(* Vertikale Linie zeichnen *)
IF Iin_X1 = Iin_X2 THEN
	in_Offset_1 := (Iin_Y1 * 80) + Iin_X1;
	FOR in_ROW_Index := Iin_Y1 TO Iin_Y2 DO
		by_old_Char := Xus_TN_SCREEN.bya_CHAR[in_Offset_1]; (* bestehendes Zeichen auslesen *)
		by_Char := by_Vertikal_Line_Char; (* Standardzeichen vorbelegen *)
		IF by_old_Char = by_Horzontal_Line_Char THEN (* Schnittpunkt erkannt *)
			IF in_ROW_Index = Iin_Y1 THEN (* Anfang der Linie behandeln *)
				by_Char := by_Connect_Top_Char;
			ELSIF in_ROW_Index = Iin_Y2 THEN (* Ende der Linie behandeln *)
				by_Char := by_Connect_Bottom_Char;
			ELSE (* Kreuzungspunkt behandeln *)
				by_Char := by_Connect_Cruz_Char;
			END_IF;
		END_IF;
		Xus_TN_SCREEN.bya_Line_Update[in_ROW_Index] := TRUE; (* Zeile zum Updaten freigeben *)
		Xus_TN_SCREEN.bya_CHAR[in_Offset_1] := by_Char;
		Xus_TN_SCREEN.bya_COLOR[in_Offset_1] := Iby_Attr;
		in_Offset_1 := in_Offset_1 + 80;
	END_FOR;

ELSIF Iin_Y1 = Iin_Y2 THEN (* Horzontale Linie zeichnen *)
	Xus_TN_SCREEN.bya_Line_Update[Iin_Y1] := TRUE; (* Zeile zum Updaten freigeben *)
	in_Offset_1 := (Iin_Y1 * 80) + Iin_X1;
	FOR in_COL_Index := Iin_X1 TO Iin_X2 DO
		by_old_Char := Xus_TN_SCREEN.bya_CHAR[in_Offset_1]; (* bestehendes Zeichen auslesen *)
		by_Char := by_Horzontal_Line_Char; (* Standardzeichen vorbelegen *)
		IF by_old_Char = by_Vertikal_Line_Char THEN (* Schnittpunkt erkannt *)
			IF in_COL_Index = Iin_X1 THEN (* Anfang der Linie behandeln *)
				by_Char := by_Connect_Left_Char;
			ELSIF in_COL_Index = Iin_X2 THEN (* Ende der Linie behandeln *)
				by_Char := by_Connect_Right_Char;
			ELSE (* Kreuzungspunkt behandeln *)
				by_Char := by_Connect_Cruz_Char;
			END_IF;
		END_IF;
		Xus_TN_SCREEN.bya_CHAR[in_Offset_1] := by_Char;
		Xus_TN_SCREEN.bya_COLOR[in_Offset_1] := Iby_Attr;
		in_Offset_1 := in_Offset_1 + 1;
	END_FOR;
END_IF;

(* revision history
ks	10. mai. 2010	rev 1.0
	original version
*)
END_FUNCTION_BLOCK

(* POU TN_SC_ADD_SHADOW, ST *)
FUNCTION_BLOCK TN_SC_ADD_SHADOW
VAR
	in_Offset : INT;
	in_X : INT;
	in_Y : INT;
END_VAR
VAR_INPUT
	Iin_Y1 : INT;
	Iin_X1 : INT;
	Iin_Y2 : INT;
	Iin_X2 : INT;
	Iin_OPTION : INT;
END_VAR
VAR_IN_OUT
	Xus_TN_SCREEN : us_TN_SCREEN;
END_VAR

(*
version 1.0		10. mai 2010
programmer		ks
tested by		ks

TN_SC_ADD_SHADOW zeichnet auf der linken und unteren Seite eines rechteckigen Bereiches einen Schatten
*)
IF TN_SC_XY2_ERROR(Iin_X1,Iin_Y1,Iin_X2,Iin_Y2) THEN RETURN; END_IF;

IF Iin_Y1 < 0 OR Iin_X1 < 0 OR Iin_Y2 < 0 OR Iin_X2 < 0 THEN RETURN; END_IF; (* min werte prüfen *)
IF Iin_Y1 > 23 OR Iin_X1 > 79 OR Iin_Y2 > 23 OR Iin_X2 > 79 THEN RETURN; END_IF; (* max werte prüfen *)

in_Offset := (Iin_Y1 * 80) + Iin_X2;

IF Iin_OPTION = INT#00 THEN
	(* Schatten durch Farbanpassung erzeugen *)
	FOR in_Y := Iin_Y1 TO Iin_Y2 DO
		Xus_TN_SCREEN.bya_COLOR[in_Offset] := TN_SC_SHADOW_ATTR(Xus_TN_SCREEN.bya_COLOR[in_Offset]);
		in_Offset := in_Offset + 80;
		Xus_TN_SCREEN.bya_Line_Update[in_Y] := TRUE; (* Zeile für Update eintragen *)
	END_FOR;
ELSE
	(* Schatten durch Farbe Schwarz und Leerzeichen erzeugen *)
	FOR in_Y := Iin_Y1 TO Iin_Y2 DO
		Xus_TN_SCREEN.bya_COLOR[in_Offset] := BYTE#00;
		Xus_TN_SCREEN.bya_CHAR[in_Offset] := BYTE#32;
		in_Offset := in_Offset + 80;
		Xus_TN_SCREEN.bya_Line_Update[in_Y] := TRUE; (* Zeile für Update eintragen *)
	END_FOR;
END_IF;

in_Offset := (Iin_Y2 * 80) + Iin_X1;

IF Iin_OPTION = INT#00 THEN
	(* Schatten durch Farbanpassung erzeugen *)
	FOR in_X  := Iin_X1 TO Iin_X2 DO
		Xus_TN_SCREEN.bya_COLOR[in_Offset] := TN_SC_SHADOW_ATTR(Xus_TN_SCREEN.bya_COLOR[in_Offset]);
		in_Offset := in_Offset + 1;
	END_FOR;
ELSE
	(* Schatten durch Farbe Schwarz und Leerzeichen erzeugen *)
	FOR in_X  := Iin_X1 TO Iin_X2 DO
		Xus_TN_SCREEN.bya_COLOR[in_Offset] := BYTE#00;
		Xus_TN_SCREEN.bya_CHAR[in_Offset] := BYTE#32;
		in_Offset := in_Offset + 1;
	END_FOR;
END_IF;

(* revision history
ks	10. mai. 2010	rev 1.0
	original version
*)
END_FUNCTION_BLOCK

(* POU TN_SC_SHADOW_ATTR, ST *)
FUNCTION TN_SC_SHADOW_ATTR : BYTE
VAR_INPUT
	Iby_ATTR : BYTE;
END_VAR

(*
version 1.0		10. mai 2010
programmer		ks
tested by		ks

TN_SC_SHADOW_ATTR berechnet aus einem normalen einem abgedunkelten Farbcode
*)
(* Background Farbe auf Schwarz ändern      *)
(* und dunkle Fordergrundfarben einschalten *)  
TN_SC_SHADOW_ATTR := ((Iby_ATTR AND BYTE#2#11110000) OR BYTE#2#00001000);

(* revision history
ks	10. mai. 2010	rev 1.0
	original version
*)
END_FUNCTION

(* POU TN_SC_BOX, ST *)
FUNCTION_BLOCK TN_SC_BOX
VAR
	FB_TN_SC_FILL : TN_SC_FILL;
	by_BorderChar_L_T : BYTE;
	by_BorderChar_T : BYTE;
	by_BorderChar_B : BYTE;
	by_BorderChar_R_T : BYTE;
	by_BorderChar_L : BYTE;
	by_BorderChar_R : BYTE;
	by_BorderChar_L_B : BYTE;
	by_BorderChar_R_B : BYTE;
	in_Y : INT;
	in_X : INT;
	in_Border_Offset : INT;
	in_Offset_1 : INT;
	in_Offset_2 : INT;
END_VAR
VAR_INPUT
	Iin_Y1 : INT;
	Iin_X1 : INT;
	Iin_Y2 : INT;
	Iin_X2 : INT;
	Iby_FILL : BYTE;
	Iby_ATTR : BYTE;
	Iin_BORDER : INT;
END_VAR
VAR_IN_OUT
	Xus_TN_SCREEN : us_TN_SCREEN;
END_VAR

(*
version 1.0		10. mai 2010
programmer		ks
tested by		ks

TN_SC_BOX füllt einen rechteckigen Bereich mit einem Zeichen und zeichnet eine Umrandung
*)
IF TN_SC_XY2_ERROR(Iin_X1,Iin_Y1,Iin_X2,Iin_Y2) THEN RETURN; END_IF;

(* Bordertype bestimmen *)
CASE Iin_Border OF
0:
	in_Border_Offset := 0;
1:
	by_BorderChar_L_T := BYTE#218; (* links oben *)
	by_BorderChar_T := BYTE#196; (* oben *)
	by_BorderChar_R_T := BYTE#191; (* rechts oben *)
	by_BorderChar_L := BYTE#179; (* links *)
	by_BorderChar_R := BYTE#179; (* rechts *)
	by_BorderChar_B := BYTE#196; (* unten *)
	by_BorderChar_L_B := BYTE#217; (* links unten *)
	by_BorderChar_R_B := BYTE#192; (* rechts unten *)
	in_Border_Offset := 1;
 2:
	by_BorderChar_L_T := BYTE#201;
	by_BorderChar_T := BYTE#205;
	by_BorderChar_R_T := BYTE#187;
	by_BorderChar_L := BYTE#186;
	by_BorderChar_R := BYTE#186;
	by_BorderChar_B := BYTE#205;
	by_BorderChar_L_B := BYTE#188;
	by_BorderChar_R_B := BYTE#200;
	in_Border_Offset := 1;
ELSE
	by_BorderChar_L_T := BYTE#32;
	by_BorderChar_T := BYTE#32;
	by_BorderChar_R_T := BYTE#32;
	by_BorderChar_L := BYTE#32;
	by_BorderChar_R := BYTE#32;
	by_BorderChar_B := BYTE#32;
	by_BorderChar_L_B := BYTE#32;
	by_BorderChar_R_B := BYTE#32;
	in_Border_Offset := 1;

END_CASE;

IF Iby_FILL > BYTE#0 THEN (* FILL Zeichen vorhanden ? -> Box zeichnen *)

	(* Fill-Function um eine Zeichenreihe kleiner zeichnen *)
	FB_TN_SC_FILL(	Iin_Y1 := Iin_Y1 + in_Border_Offset,
					Iin_X1 := Iin_X1 + in_Border_Offset,
					Iin_Y2 := Iin_Y2 - in_Border_Offset,
					Iin_X2 := Iin_X2 - in_Border_Offset,
					Iby_CHAR := Iby_FILL,
					Iby_Attr := Iby_ATTR,
					Xus_TN_SCREEN := Xus_TN_SCREEN);
END_IF;

IF Iin_BORDER = 0 THEN RETURN; END_IF;

(* linken und rechten Rand ausgeben *)

in_Offset_1 := (Iin_Y1 * 80) + Iin_X1;
in_Offset_2 := (Iin_Y1 * 80) + Iin_X2;

FOR in_Y := Iin_Y1 TO Iin_Y2 DO

	(* Zeile zum Updaten freigeben *)
	Xus_TN_SCREEN.bya_Line_Update[in_Y] := TRUE;

	Xus_TN_SCREEN.bya_CHAR[in_Offset_1] := by_BorderChar_L;
	Xus_TN_SCREEN.bya_COLOR[in_Offset_1] := Iby_Attr;

	Xus_TN_SCREEN.bya_CHAR[in_Offset_2] := by_BorderChar_R;
	Xus_TN_SCREEN.bya_COLOR[in_Offset_2] := Iby_Attr;

	in_Offset_1 := in_Offset_1 + 80;
	in_Offset_2 := in_Offset_2 + 80;

END_FOR;

(* unteren und oberen Rand ausgeben *)
in_Offset_1 := (Iin_Y1 * 80) + Iin_X1;
in_Offset_2 := (Iin_Y2 * 80) + Iin_X1;

FOR in_X := Iin_X1 TO Iin_X2 DO

	Xus_TN_SCREEN.bya_CHAR[in_Offset_1] := by_BorderChar_T;
	Xus_TN_SCREEN.bya_COLOR[in_Offset_1] := Iby_Attr;

	Xus_TN_SCREEN.bya_CHAR[in_Offset_2] := by_BorderChar_B;
	Xus_TN_SCREEN.bya_COLOR[in_Offset_2] := Iby_Attr;

	in_Offset_1 := in_Offset_1 + INT#1;
	in_Offset_2 := in_Offset_2 + INT#1;

END_FOR;

(* linke obere Ecke ausgeben *)
in_Offset_1 := (Iin_Y1 * 80) + Iin_X1;
Xus_TN_SCREEN.bya_CHAR[in_Offset_1] := by_BorderChar_L_T;
Xus_TN_SCREEN.bya_COLOR[in_Offset_1] := Iby_Attr;

(* rechte obere Ecke ausgeben *)
in_Offset_1 := (Iin_Y1 * 80) + Iin_X2;
Xus_TN_SCREEN.bya_CHAR[in_Offset_1] := by_BorderChar_R_T;
Xus_TN_SCREEN.bya_COLOR[in_Offset_1] := Iby_Attr;

(* linke untere Ecke ausgeben *)
in_Offset_1 := (Iin_Y2 * 80) + Iin_X1;
Xus_TN_SCREEN.bya_CHAR[in_Offset_1] := by_BorderChar_R_B;
Xus_TN_SCREEN.bya_COLOR[in_Offset_1] := Iby_Attr;

(* rechte untere Ecke ausgeben *)
in_Offset_1 := (Iin_Y2 * 80) + Iin_X2;
Xus_TN_SCREEN.bya_CHAR[in_Offset_1] := by_BorderChar_L_B;
Xus_TN_SCREEN.bya_COLOR[in_Offset_1] := Iby_Attr;

(* revision history
ks	10. mai. 2010	rev 1.0
	original version
*)
END_FUNCTION_BLOCK

(* POU TN_SC_FILL, ST *)
FUNCTION_BLOCK TN_SC_FILL
VAR
	in_X : INT;
	in_Y : INT;
	in_Offset : INT;
END_VAR
VAR_INPUT
	Iin_Y1 : INT;
	Iin_X1 : INT;
	Iin_Y2 : INT;
	Iin_X2 : INT;
	Iby_CHAR : BYTE;
	Iby_Attr : BYTE;
END_VAR
VAR_IN_OUT
	Xus_TN_SCREEN : us_TN_SCREEN;
END_VAR

(*
version 1.0		10. mai 2010
programmer		ks
tested by		ks

TN_SC_FILL füllt einen rechteckigen Bereich mit einem Zeichen
*)
IF TN_SC_XY2_ERROR(Iin_X1,Iin_Y1,Iin_X2,Iin_Y2) THEN RETURN; END_IF;

FOR in_Y := Iin_Y1 TO Iin_Y2 DO
	Xus_TN_SCREEN.bya_Line_Update[in_Y] := TRUE; (* Zeile zum Updaten freigeben *)
	in_Offset := (in_Y * 80) + Iin_X1;
	FOR in_X := Iin_X1 TO Iin_X2 DO
		Xus_TN_SCREEN.bya_CHAR[in_Offset]  := Iby_CHAR; (* Zeichen eintragen *)
		Xus_TN_SCREEN.bya_COLOR[in_Offset] := Iby_Attr; (* Farbe eintragen *)
		in_Offset := in_Offset + 1;
	END_FOR;
END_FOR;

(* revision history
ks	10. mai. 2010	rev 1.0
	original version
*)
END_FUNCTION_BLOCK

(* POU TN_SC_WRITE_C, ST *)
FUNCTION_BLOCK TN_SC_WRITE_C
VAR
	FB_TN_SC_WRITE : TN_SC_WRITE;
END_VAR
VAR_INPUT
	Iin_Y : INT;
	Iin_X : INT;
	Iby_ATTR : BYTE;
	Ist_STRING : STRING;
	Iin_LENGTH : INT;
	Iin_OPTION : INT;
END_VAR
VAR_IN_OUT
	Xus_TN_SCREEN : us_TN_SCREEN;
END_VAR

(*
version 1.0		10. mai 2010
programmer		ks
tested by		ks

TN_SC_WRITE_C korrigiert die Textlänge und schreibt den Text an die angegebenen Koordinate
*)
(* Text ausgeben *)
FB_TN_SC_WRITE( Iin_Y := Iin_Y,
				Iin_X := Iin_X,
				Iby_ATTR := Iby_ATTR,
				Ist_STRING := FIX(str:=Ist_STRING,L:=Iin_LENGTH,C:=BYTE#32,M:=Iin_OPTION),
				Xus_TN_SCREEN := Xus_TN_SCREEN);

(* revision history
ks	10. mai. 2010	rev 1.0
	original version
*)
END_FUNCTION_BLOCK

(* POU TN_SC_WRITE, ST *)
FUNCTION_BLOCK TN_SC_WRITE
VAR
	bo_Color : BOOL;
	in_Offset : INT;
	in_Char_Index : INT;
	in_String_Length : INT;
END_VAR
VAR_INPUT
	Iin_Y : INT;
	Iin_X : INT;
	Iby_ATTR : BYTE;
	Ist_STRING : STRING;
END_VAR
VAR_IN_OUT
	Xus_TN_SCREEN : us_TN_SCREEN;
END_VAR

(*
version 1.0		10. mai 2010
programmer		ks
tested by		ks

TN_SC_WRITE schreibt einem Text an die angegebene Koordinate
*)
in_String_Length := LEN(Ist_STRING);
IF TN_SC_XY_ERROR(Iin_X + in_String_Length - 1,Iin_Y) THEN RETURN; END_IF;
Xus_TN_SCREEN.bya_Line_Update[Iin_Y] := TRUE; (* Zeile zum Updaten freigeben *)
in_Offset := (Iin_Y * 80) + Iin_X; (* Offset des ersten Zeichen berechnen *)
bo_Color := Iby_ATTR <> BYTE#00;

(* Zeichen und Attribute des String kopieren *)
FOR in_Char_Index := 1 TO in_String_Length DO
	IF bo_Color THEN Xus_TN_SCREEN.bya_COLOR[in_Offset] := Iby_ATTR; END_IF;
	Xus_TN_SCREEN.bya_CHAR[in_Offset] := CODE(STR:=Ist_STRING,POS:=in_Char_Index);
	in_Offset := in_Offset + INT#1;
END_FOR;

Xus_TN_SCREEN.in_EOS_Offset := in_Offset; (* End of String Offset sichern *)

(* revision history
ks	10. mai. 2010	rev 1.0
	original version
*)
END_FUNCTION_BLOCK

(* POU TN_SC_XY_ERROR, ST *)
FUNCTION TN_SC_XY_ERROR : BOOL
VAR_INPUT
	X : INT;
	Y : INT;
END_VAR

(*
version 1.0		10. mai 2010
programmer		ks
tested by		ks

TN_SC_XY_ERROR prüft ob die angegenene Koordinaten gültig sind 
*)
(* min und max werte prüfen *)
TN_SC_XY_ERROR := Y < 0 OR X < 0 OR Y > 23 OR X > 79;

(* revision history
ks	10. mai. 2010	rev 1.0
	original version
*)
END_FUNCTION

(* POU TN_INPUT_SELECT_TEXT, ST *)
FUNCTION_BLOCK TN_INPUT_SELECT_TEXT
VAR
	in_count : INT;
	by_Attr : BYTE;
	st_String : STRING;
END_VAR
VAR
	FB_TN_SC_WRITE : TN_SC_WRITE;
END_VAR
VAR_IN_OUT
	Xus_TN_SCREEN : us_TN_SCREEN;
	Xus_TN_INPUT_CONTROL_DATA : us_TN_INPUT_CONTROL_DATA;
END_VAR

(*
version 1.1		06. apr 2011
programmer		ks
tested by			ks

TN_SELECT_TEXT dient zur verwaltung und darstellung einer Elementeauswahl
*)
(* Benutzereingabe auswerten -> Selektion Text n *)
IF Xus_TN_INPUT_CONTROL_DATA.bo_Focus = TRUE THEN

(* Leertaste-Taste auswerten *)
	IF Xus_TN_INPUT_CONTROL_DATA.by_Input_ASCII_Code = BYTE#32 THEN
		Xus_TN_INPUT_CONTROL_DATA.in_selected := Xus_TN_INPUT_CONTROL_DATA.in_selected + INT#01; 
		Xus_TN_INPUT_CONTROL_DATA.bo_Update_Input := TRUE;
	END_IF;
 
	(* Return-Taste auswerten *)
	IF Xus_TN_INPUT_CONTROL_DATA.by_Input_Exten_Code = BYTE#13 THEN
		Xus_TN_INPUT_CONTROL_DATA.bo_Input_Entered := TRUE;
	END_IF;

END_IF;

(* Aktualisierung der Anzeige *)
IF (Xus_TN_INPUT_CONTROL_DATA.bo_Update_Input = TRUE) OR (Xus_TN_INPUT_CONTROL_DATA.bo_Update_All = TRUE) THEN

	(* Title-Text ausgeben *)
	IF Xus_TN_INPUT_CONTROL_DATA.bo_Update_All = TRUE THEN

		IF (Xus_TN_INPUT_CONTROL_DATA.in_Title_X_Offset = INT#00) AND (Xus_TN_INPUT_CONTROL_DATA.in_Title_Y_Offset = INT#00) THEN
			(* wenn Offset X,Y =0 dann Titlestring links vom Element positionieren *)
			FB_TN_SC_WRITE.Iin_Y := Xus_TN_INPUT_CONTROL_DATA.in_Y;
			FB_TN_SC_WRITE.Iin_X := Xus_TN_INPUT_CONTROL_DATA.in_X - LEN(Xus_TN_INPUT_CONTROL_DATA.st_Title_String);

		ELSE
			(* Title-Text durch Row, Color-Offset ausgeben *)
			FB_TN_SC_WRITE.Iin_Y := Xus_TN_INPUT_CONTROL_DATA.in_Y + Xus_TN_INPUT_CONTROL_DATA.in_Title_Y_Offset;
			FB_TN_SC_WRITE.Iin_X := Xus_TN_INPUT_CONTROL_DATA.in_X + Xus_TN_INPUT_CONTROL_DATA.in_Title_X_Offset;
		END_IF;

		(* Title-Text durch Row, Color-Offset ausgeben *)
		FB_TN_SC_WRITE(	Iby_ATTR := Xus_TN_INPUT_CONTROL_DATA.by_Title_Attr,
						Ist_STRING := Xus_TN_INPUT_CONTROL_DATA.st_Title_String,
						Xus_TN_SCREEN := Xus_TN_SCREEN);

	END_IF;

	(* Eingabezeile verarbeiten *)

	(* Anzahl der Elemente bestimmen *)
	in_count := ELEMENT_COUNT(SEP:=BYTE#35,ELEMENT:=Xus_TN_INPUT_CONTROL_DATA.st_Input_Data);

	IF in_Count > INT#00 THEN

		IF Xus_TN_INPUT_CONTROL_DATA.in_selected < INT#1 THEN
			Xus_TN_INPUT_CONTROL_DATA.in_selected := INT#01;
		END_IF;

		IF Xus_TN_INPUT_CONTROL_DATA.in_selected > in_count THEN
			Xus_TN_INPUT_CONTROL_DATA.in_selected := INT#01;
		END_IF;

		st_String := ELEMENT_GET(SEP:=BYTE#35,POS:=Xus_TN_INPUT_CONTROL_DATA.in_selected - 1,ELEMENT:=Xus_TN_INPUT_CONTROL_DATA.st_Input_Data);

		st_String := FIX(	str:=st_String,
							L:=LEN(Xus_TN_INPUT_CONTROL_DATA.st_Input_Mask),
							C:=BYTE#32,
							M:=Xus_TN_INPUT_CONTROL_DATA.in_Input_Option);

		Xus_TN_INPUT_CONTROL_DATA.st_Input_String := st_String;

		IF Xus_TN_INPUT_CONTROL_DATA.bo_Focus = TRUE THEN
			by_Attr := Xus_TN_INPUT_CONTROL_DATA.by_Attr_mF;
		ELSE
			by_Attr := Xus_TN_INPUT_CONTROL_DATA.by_Attr_oF;
		END_IF;

		FB_TN_SC_WRITE(	Iin_Y := Xus_TN_INPUT_CONTROL_DATA.in_Y,
						Iin_X := Xus_TN_INPUT_CONTROL_DATA.in_X,
						Iby_ATTR := by_Attr,
						Ist_STRING := st_String,
						Xus_TN_SCREEN := Xus_TN_SCREEN);
	END_IF;

	(* Cursor auf aktuelle Position setzen *)
	Xus_TN_INPUT_CONTROL_DATA.in_Cursor_Y := Xus_TN_INPUT_CONTROL_DATA.in_Y;
	Xus_TN_INPUT_CONTROL_DATA.in_Cursor_X := Xus_TN_INPUT_CONTROL_DATA.in_X;

	(* Update-Flag's rücksetzen *)
	Xus_TN_INPUT_CONTROL_DATA.bo_Update_All := FALSE;
	Xus_TN_INPUT_CONTROL_DATA.bo_Update_Input := FALSE;

END_IF;

(* revision history

ks	06. apr. 2011	rev 1.1
	list_len und list_get durch element_count und element_get ersetzt

ks	10. mai. 2010	rev 1.0
	original version
*)
END_FUNCTION_BLOCK

(* POU TN_INPUT_EDIT_LINE, ST *)
FUNCTION_BLOCK TN_INPUT_EDIT_LINE
VAR
	in_count : INT;
	in_Count_End : INT;
	in_CursorOffset : INT;
	by_Attr : BYTE;
	st_String : STRING;
	bo_Pos_Found : BOOL;
	st_CHAR : STRING(1);
	in_old_charpos : INT;
END_VAR
VAR
	FB_TN_SC_WRITE : TN_SC_WRITE;
END_VAR
VAR_IN_OUT
	Xus_TN_SCREEN : us_TN_SCREEN;
	Xus_TN_INPUT_CONTROL_DATA : us_TN_INPUT_CONTROL_DATA;
END_VAR

(*
version 1.0		10. mai 2010
programmer		ks
tested by		ks

TN_INPUT_EDIT_LINE ermöglicht die Eingabe von Texten durch eine Editierbare Eingabezeile
*)
(* Cursorsteuerung rücksetzen *)
in_CursorOffset := INT#0;

IF Xus_TN_INPUT_CONTROL_DATA.bo_Focus = TRUE THEN

	(* Texteingabe erkannt ? *)
	IF Xus_TN_INPUT_CONTROL_DATA.by_Input_ASCII_Code > BYTE#0 THEN

		IF (Xus_TN_INPUT_CONTROL_DATA.bo_Input_Only_Num = TRUE AND Xus_TN_INPUT_CONTROL_DATA.bo_Input_ASCII_IsNum = TRUE)
			OR (Xus_TN_INPUT_CONTROL_DATA.bo_Input_Only_Num = FALSE) THEN

			(* ASCII Wert in einen String wandeln *)
			st_CHAR := CHR_TO_STRING(C:=Xus_TN_INPUT_CONTROL_DATA.by_Input_ASCII_Code);

			(* Eingabe übernehmen *)
			Xus_TN_INPUT_CONTROL_DATA.st_Input_Data := REPLACE(Xus_TN_INPUT_CONTROL_DATA.st_Input_Data,
			st_CHAR,INT#1,Xus_TN_INPUT_CONTROL_DATA.in_Cursor_Pos);

			in_CursorOffset := INT#1;
			Xus_TN_INPUT_CONTROL_DATA.bo_Update_Input := TRUE;
		END_IF;
	END_IF;

	CASE BYTE_TO_INT(Xus_TN_INPUT_CONTROL_DATA.by_Input_Exten_Code) OF

	67: (* Cursor rechts gedrückt *)
		in_CursorOffset := INT#1;

	68: (* Cursor links gedrückt *)
		in_CursorOffset := -1;

	08: (* Backspace gedrückt *)
		Xus_TN_INPUT_CONTROL_DATA.st_Input_Data := REPLACE(Xus_TN_INPUT_CONTROL_DATA.st_Input_Data, ' ', 1,Xus_TN_INPUT_CONTROL_DATA.in_Cursor_Pos);
		Xus_TN_INPUT_CONTROL_DATA.bo_Update_Input := TRUE;
		in_CursorOffset := -1;

	13: (* Enter-Taste gedrückt *)
		IF LEN(Xus_TN_INPUT_CONTROL_DATA.st_Input_Mask) > INT#00 THEN
			(* Eingabestring übernehmen *)
			Xus_TN_INPUT_CONTROL_DATA.st_Input_String := Xus_TN_INPUT_CONTROL_DATA.st_Input_Data;

			(* Eingabestring -> links und rechts Leerzeichen entfernen *)
			Xus_TN_INPUT_CONTROL_DATA.st_Input_String := TRIME(str:=Xus_TN_INPUT_CONTROL_DATA.st_Input_String);
			Xus_TN_INPUT_CONTROL_DATA.bo_Input_Entered := TRUE;

			(* neue Eingabe vorbereiten *)
			Xus_TN_INPUT_CONTROL_DATA.st_Input_Data := Xus_TN_INPUT_CONTROL_DATA.st_Input_Mask;

			Xus_TN_INPUT_CONTROL_DATA.in_Cursor_Pos := INT#1;
			Xus_TN_INPUT_CONTROL_DATA.bo_Update_Input := TRUE;

			(* suche erstes Position in Eingabemaske *)
			st_CHAR := MID(Xus_TN_INPUT_CONTROL_DATA.st_Input_Mask,1,Xus_TN_INPUT_CONTROL_DATA.in_Cursor_Pos);
			IF st_CHAR <> ' ' THEN
				(* nächsten Eingabeposition suchen *)
				in_CursorOffset := INT#1;
			END_IF;
		END_IF;
	END_CASE;
END_IF;

(* Cursor richtung rechts bewegen                                   *)
IF (in_CursorOffset > INT#0) OR (Xus_TN_INPUT_CONTROL_DATA.in_Cursor_Pos = INT#0) THEN
	bo_Pos_Found := FALSE;

	in_Count := Xus_TN_INPUT_CONTROL_DATA.in_Cursor_Pos + INT#1;
	in_Count_End := LEN(Xus_TN_INPUT_CONTROL_DATA.st_Input_Mask);

	WHILE (in_count <= in_Count_End) AND (bo_Pos_Found = FALSE) DO

		st_CHAR := MID(Xus_TN_INPUT_CONTROL_DATA.st_Input_Mask,1,in_count);
		IF st_CHAR = ' ' THEN
			Xus_TN_INPUT_CONTROL_DATA.in_Cursor_Pos := in_count;
			Xus_TN_INPUT_CONTROL_DATA.bo_Update_Input := TRUE;
			bo_Pos_Found := TRUE;
		END_IF;

		in_count := in_count + INT#1;

	END_WHILE;
END_IF;

(* Cursor richtung links bewegen *)
IF in_CursorOffset < INT#0 THEN
	bo_Pos_Found := FALSE;

	in_Count     := Xus_TN_INPUT_CONTROL_DATA.in_Cursor_Pos - INT#01;
	in_Count_End := INT#1;

	WHILE (in_count >= in_Count_End) AND (bo_Pos_Found = FALSE) DO

		st_CHAR := MID(Xus_TN_INPUT_CONTROL_DATA.st_Input_Mask,1,in_count);
		IF st_CHAR = ' ' THEN
			Xus_TN_INPUT_CONTROL_DATA.in_Cursor_Pos := in_count;
			Xus_TN_INPUT_CONTROL_DATA.bo_Update_Input := TRUE;
			bo_Pos_Found := TRUE;
		END_IF;

		in_count := in_count - INT#1;
	END_WHILE;
END_IF;

(* maximale Cursorposition ? *)
IF Xus_TN_INPUT_CONTROL_DATA.in_Cursor_Pos > LEN(Xus_TN_INPUT_CONTROL_DATA.st_Input_Data) THEN
	Xus_TN_INPUT_CONTROL_DATA.in_Cursor_Pos := LEN(Xus_TN_INPUT_CONTROL_DATA.st_Input_Data);
	Xus_TN_INPUT_CONTROL_DATA.bo_Update_Input := TRUE;
END_IF;

(* minimale Cursorposition ? *)
IF Xus_TN_INPUT_CONTROL_DATA.in_Cursor_Pos < INT#1 THEN
	Xus_TN_INPUT_CONTROL_DATA.in_Cursor_Pos := INT#1;
	Xus_TN_INPUT_CONTROL_DATA.bo_Update_Input := TRUE;
END_IF;

(* Aktualisierung der Anzeige *)
IF (Xus_TN_INPUT_CONTROL_DATA.bo_Update_Input = TRUE) OR (Xus_TN_INPUT_CONTROL_DATA.bo_Update_All = TRUE) THEN

	(* Title-Text ausgeben *)
	IF (Xus_TN_INPUT_CONTROL_DATA.bo_Update_All = TRUE) THEN

		IF (Xus_TN_INPUT_CONTROL_DATA.in_Title_X_Offset = INT#00) AND (Xus_TN_INPUT_CONTROL_DATA.in_Title_Y_Offset = INT#00) THEN
			(* wenn Offset X,Y =0 dann Titlestring links vom Element positionieren *)
			FB_TN_SC_WRITE.Iin_Y := Xus_TN_INPUT_CONTROL_DATA.in_Y;
			FB_TN_SC_WRITE.Iin_X := Xus_TN_INPUT_CONTROL_DATA.in_X - LEN(Xus_TN_INPUT_CONTROL_DATA.st_Title_String);
		ELSE
			(* Title-Text durch Row, Color-Offset ausgeben *)
			FB_TN_SC_WRITE.Iin_Y := Xus_TN_INPUT_CONTROL_DATA.in_Y + Xus_TN_INPUT_CONTROL_DATA.in_Title_Y_Offset;
			FB_TN_SC_WRITE.Iin_X := Xus_TN_INPUT_CONTROL_DATA.in_X + Xus_TN_INPUT_CONTROL_DATA.in_Title_X_Offset;
		END_IF;

		(* Title-Text durch Row, Color-Offset ausgeben *)
		FB_TN_SC_WRITE(	Iby_ATTR := Xus_TN_INPUT_CONTROL_DATA.by_Title_Attr,
						Ist_STRING := Xus_TN_INPUT_CONTROL_DATA.st_Title_String,
						Xus_TN_SCREEN := Xus_TN_SCREEN);
	END_IF;

	(* Eingabetext ausgeben *)
	IF (Xus_TN_INPUT_CONTROL_DATA.bo_Input_Hidden = TRUE) THEN

		st_String := '';

		IF LEN(Xus_TN_INPUT_CONTROL_DATA.st_Input_Data) = LEN(Xus_TN_INPUT_CONTROL_DATA.st_Input_Mask) THEN
			(* Eingabemodus: HIDDEN *)
			FOR in_count := 1 TO LEN(Xus_TN_INPUT_CONTROL_DATA.st_Input_Data) DO

				(* Zeichen aus Eingabemaske lesen *)
				st_CHAR := MID(Xus_TN_INPUT_CONTROL_DATA.st_Input_Mask,1,in_count);

				(* Eingabe oder Maskenzeichen ausgeben *)
				IF st_CHAR = ' ' THEN

					(* Zeichen aus Eingabedata lesen *)
					st_CHAR := MID(Xus_TN_INPUT_CONTROL_DATA.st_Input_Data,1,in_count);

					IF st_CHAR = ' ' THEN
						(* Leerzeichen ausgeben *)
						st_String := CONCAT(st_String, ' ');

					ELSE
						(* verdecktes Zeichen ausgeben *)
						st_String := CONCAT(st_String, '*');

					END_IF;

				ELSE
					(* Zeichen aus Eingabemaske übernehmen *)
					st_CHAR := MID(Xus_TN_INPUT_CONTROL_DATA.st_Input_Data,1,in_count);
					st_String := CONCAT(st_String,st_CHAR);

				END_IF;
			END_FOR;
		END_IF;
	ELSE

		(* Eingabemodus: NORMAL *)
		st_String := Xus_TN_INPUT_CONTROL_DATA.st_Input_Data;

	END_IF;

	(* String ausgeben *)

	IF Xus_TN_INPUT_CONTROL_DATA.bo_Focus = TRUE THEN
		by_Attr := Xus_TN_INPUT_CONTROL_DATA.by_Attr_mF;
	ELSE
		by_Attr := Xus_TN_INPUT_CONTROL_DATA.by_Attr_oF;
	END_IF;

	FB_TN_SC_WRITE(	Iin_Y := Xus_TN_INPUT_CONTROL_DATA.in_Y,
					Iin_X := Xus_TN_INPUT_CONTROL_DATA.in_X,
					Iby_ATTR := by_Attr,
					Ist_STRING := st_String,
					Xus_TN_SCREEN := Xus_TN_SCREEN);

	(* Cursor auf aktuelle Position setzen *)
	Xus_TN_INPUT_CONTROL_DATA.in_Cursor_Y := Xus_TN_INPUT_CONTROL_DATA.in_Y;
	Xus_TN_INPUT_CONTROL_DATA.in_Cursor_X := Xus_TN_INPUT_CONTROL_DATA.in_X + Xus_TN_INPUT_CONTROL_DATA.in_Cursor_Pos - INT#1;

	in_old_charpos := INT#0;

	(* Update-Flag's rücksetzen *)
	Xus_TN_INPUT_CONTROL_DATA.bo_Update_All := FALSE;
	Xus_TN_INPUT_CONTROL_DATA.bo_Update_Input := FALSE;
END_IF;

(* revision history
ks	10. mai. 2010	rev 1.0
	original version
*)
END_FUNCTION_BLOCK

(* POU TN_INPUT_MENU_BAR, ST *)
FUNCTION_BLOCK TN_INPUT_MENU_BAR
VAR
	FB_TN_INPUT_MENU_POPUP : TN_INPUT_MENU_POPUP;
	us_TN_MENU_POPUP : us_TN_MENU_POPUP;
	FB_TN_SC_WRITE_C : TN_SC_WRITE_C;
END_VAR
VAR
	in_ROW : INT;
	in_COL : INT;
	in_TITLE_Length : INT;
	st_MENU_BAR : STRING(STRING_LENGTH);
	st_MENU_TITLE : STRING;
	in_Count : INT;
	in_Index : INT;
	by_New_KeyCode : BYTE;
	in_Scroll_Offset : INT;
	by_ATTR : BYTE;
	bo_Reset_Position :	BOOL;
END_VAR
VAR_IN_OUT
	Xus_TN_MENU : us_TN_MENU;
	Xus_TN_SCREEN : us_TN_SCREEN;
END_VAR

(*
version 1.1		06. apr 2011
programmer		ks
tested by			ks

TN_MENU_BAR ermöglicht die verwaltung und darstellung einer MENU-BAR
*)
(* sicherstellen das rechteck immer innerhalb screen positioniert wird *)

IF (Xus_TN_MENU.in_State = INT#00) AND (Xus_TN_MENU.bo_Create = TRUE) THEN
	Xus_TN_MENU.in_State := INT#01;
	Xus_TN_MENU.bo_Create := FALSE;
	Xus_TN_MENU.in_Menu_Selected := INT#00;
	Xus_TN_MENU.bo_Update := TRUE;
	bo_Reset_Position := TRUE;

	(* Menu-Bar - Hauptmenue *)
	st_MENU_BAR := ELEMENT_GET(SEP:=BYTE#37,POS:=0,ELEMENT:=Xus_TN_MENU.st_MENU_TEXT);

	(* Menu-Bar - Anzahl der Elemente bestimmen *)
	Xus_TN_MENU.in_Menu_E_Count := ELEMENT_COUNT(SEP:=BYTE#35,ELEMENT:=st_MENU_BAR);

END_IF;

(* Keycode ablegen *)
by_New_KeyCode := Xus_TN_SCREEN.by_Input_Exten_Code;

(* Popup-Menu Tastensteuerung (nur Cursor oben + unten zulassen *)
IF (by_New_KeyCode = BYTE#65) OR (by_New_KeyCode = BYTE#66) THEN
	us_TN_MENU_POPUP.by_Input_Exten_Code := by_New_KeyCode;
ELSE
	us_TN_MENU_POPUP.by_Input_Exten_Code := BYTE#00;
END_IF;

(* Escape *)
IF (by_New_KeyCode = BYTE#27) THEN
	(* Menu war inaktiv -> Escape -> Menu aktivieren *)
	IF (Xus_TN_MENU.in_State = INT#01) AND (Xus_TN_SCREEN.bo_Modal_Dialog = FALSE) THEN
		Xus_TN_MENU.in_State := INT#02;
		Xus_TN_MENU.bo_Update := TRUE;
		Xus_TN_MENU.in_Menu_Selected := INT#00;

		Xus_TN_SCREEN.bo_Menue_Bar_Dialog := TRUE;

		(* Menu war aktiv -> Escape -> Menu deaktivieren *)
	ELSIF (Xus_TN_MENU.in_State = INT#02) THEN
		us_TN_MENU_POPUP.bo_Destroy := TRUE;
		Xus_TN_MENU.bo_Update := TRUE;
		Xus_TN_MENU.in_State := INT#01;
		bo_Reset_Position := TRUE;

		Xus_TN_SCREEN.bo_Menue_Bar_Dialog := FALSE;
	END_IF;
END_IF;

(* Menu aktiv *)
IF (Xus_TN_MENU.in_State = INT#02) THEN

	(* Return *)
	IF (by_New_KeyCode = BYTE#13)  THEN
		us_TN_MENU_POPUP.bo_Destroy := TRUE;
		Xus_TN_MENU.bo_Update := TRUE;
		Xus_TN_MENU.in_State := INT#01;
		bo_Reset_Position := TRUE;
		Xus_TN_MENU.in_Menu_Selected := (Xus_TN_MENU.in_Cur_Menu_Item * INT#10) + Xus_TN_MENU.in_Cur_Sub_Item;
		Xus_TN_SCREEN.by_Input_Exten_Code := BYTE#00;

		Xus_TN_SCREEN.bo_Menue_Bar_Dialog := FALSE;

		(* Destroy-Befehl -> Popup-Menu beenden *)
	ELSIF (Xus_TN_MENU.bo_Destroy = TRUE) THEN
		us_TN_MENU_POPUP.bo_Destroy := TRUE;
		Xus_TN_MENU.bo_Update := TRUE;
		Xus_TN_MENU.in_State := INT#01;
		bo_Reset_Position := TRUE;
		Xus_TN_MENU.in_Menu_Selected := INT#00;
		Xus_TN_SCREEN.by_Input_Exten_Code := BYTE#00;

		Xus_TN_SCREEN.bo_Menue_Bar_Dialog := FALSE;

	END_IF;

	IF (by_New_KeyCode = BYTE#67) THEN (* Cursor rechts *)
		in_Scroll_Offset := INT#1;
		Xus_TN_MENU.bo_Update := TRUE;
		Xus_TN_SCREEN.by_Input_Exten_Code := BYTE#00;

	ELSIF (by_New_KeyCode = BYTE#68) THEN (* Cursor links *)
		in_Scroll_Offset := -1;
		Xus_TN_MENU.bo_Update := TRUE;
		Xus_TN_SCREEN.by_Input_Exten_Code := BYTE#00;
	END_IF;
END_IF;

IF bo_Reset_Position = TRUE THEN
	bo_Reset_Position := FALSE;
	Xus_TN_MENU.in_X_SM_old := -1;
	Xus_TN_MENU.in_Y_SM_old := -1;
	Xus_TN_MENU.in_X_SM_new := -1;
	Xus_TN_MENU.in_Y_SM_new := -1;
END_IF;

(* POPUP-Menu updaten *)
IF (Xus_TN_MENU.in_State > INT#00) AND (Xus_TN_MENU.bo_Update = TRUE) THEN

	Xus_TN_MENU.bo_Update := FALSE; 

	in_ROW := Xus_TN_MENU.in_Y;
	in_COL := Xus_TN_MENU.in_X;

	(* Scrolloffset *)
	IF in_Scroll_Offset <> INT#00 THEN
		Xus_TN_MENU.in_Cur_Menu_Item := INC2(Xus_TN_MENU.in_Cur_Menu_Item,in_Scroll_Offset,1,Xus_TN_MENU.in_Menu_E_Count);
		in_Scroll_Offset := INT#00;
	ELSE
		(* Item = 0 und kein Scrolloffset *)
		IF (Xus_TN_MENU.in_Cur_Menu_Item = INT#00) THEN
			Xus_TN_MENU.in_Cur_Menu_Item := INT#01;
		END_IF;
	END_IF;

	(* alle Menutext zeichnen *)
	FOR in_Count := INT#01 TO Xus_TN_MENU.in_Menu_E_Count DO;

		(* Zeichenfarbe bestimmen *)
		IF (in_Count = Xus_TN_MENU.in_Cur_Menu_Item) AND (Xus_TN_MENU.in_State > INT#01 ) THEN
			by_ATTR := Xus_TN_MENU.by_Attr_mF;

			Xus_TN_MENU.in_Y_SM_new := in_ROW + INT#01;
			Xus_TN_MENU.in_X_SM_new := in_COL;

		ELSE
			by_ATTR := Xus_TN_MENU.by_Attr_oF;
		END_IF;

		st_MENU_TITLE := ELEMENT_GET(SEP:=BYTE#35,POS:=in_Count - 1,ELEMENT:=st_MENU_BAR);

		in_TITLE_Length := LEN(st_MENU_TITLE) + INT#02;

		FB_TN_SC_WRITE_C(	Iin_Y := in_ROW,
							Iin_X := in_COL,
							Iby_ATTR := by_ATTR,
							Iin_LENGTH := in_TITLE_Length,
							Iin_OPTION := INT#02,
							Ist_STRING := st_MENU_TITLE,
							Xus_TN_SCREEN := Xus_TN_SCREEN);

		in_COL := in_COL + in_TITLE_Length;

	END_FOR;
END_IF;

IF Xus_TN_MENU.in_X_SM_new <> Xus_TN_MENU.in_X_SM_old THEN

	(* SubMenu ist aktiv -> beenden                                     *)
	IF us_TN_MENU_POPUP.bo_Activ = TRUE THEN
		us_TN_MENU_POPUP.bo_Destroy := TRUE;

		(* Sub-Menu bearbeiten *)
		FB_TN_INPUT_MENU_POPUP(	Xus_TN_MENU_POPUP := us_TN_MENU_POPUP,
								Xus_TN_SCREEN := Xus_TN_SCREEN);
	END_IF;

	IF us_TN_MENU_POPUP.bo_Activ = FALSE THEN
		(* Popup-Menu zu aktuellen Menu parametrieren und ausführen         *)
		in_Index := Xus_TN_MENU.in_Cur_Menu_Item;

		us_TN_MENU_POPUP.in_Y := Xus_TN_MENU.in_Y_SM_new;
		us_TN_MENU_POPUP.in_X := Xus_TN_MENU.in_X_SM_new;
		us_TN_MENU_POPUP.by_Attr_mF := Xus_TN_MENU.by_Attr_mF;
		us_TN_MENU_POPUP.by_Attr_oF := Xus_TN_MENU.by_Attr_oF;
		us_TN_MENU_POPUP.st_Menu_Text := ELEMENT_GET(SEP:=BYTE#37,POS:=in_Index,ELEMENT:=Xus_TN_MENU.st_MENU_TEXT);
		us_TN_MENU_POPUP.bo_Create := TRUE;

		Xus_TN_MENU.in_X_SM_old := Xus_TN_MENU.in_X_SM_new;
		Xus_TN_MENU.in_Y_SM_old := Xus_TN_MENU.in_Y_SM_new;

	END_IF;
END_IF;

(* Popup-Menu zyklisch aufrufen *)
FB_TN_INPUT_MENU_POPUP(	Xus_TN_MENU_POPUP := us_TN_MENU_POPUP,
						Xus_TN_SCREEN := Xus_TN_SCREEN);

(* aktuelles Item vom Popup-Menu kopieren *)
Xus_TN_MENU.in_Cur_Sub_Item := us_TN_MENU_POPUP.in_Cur_Item;

(* Destroy-Befehl *)
IF (Xus_TN_MENU.in_State = INT#01) THEN
	IF (Xus_TN_MENU.bo_Destroy = TRUE) THEN
		Xus_TN_MENU.in_State := INT#00;
		Xus_TN_MENU.bo_Destroy := FALSE;
		Xus_TN_MENU.in_Cur_Menu_Item := INT#00;
		Xus_TN_MENU.in_Cur_Sub_Item := INT#00;
	END_IF;
END_IF;

(* revision history
ks	06. apr. 2011	rev 1.1
	list_len und list_get durch element_count und element_get ersetzt

ks	10. mai. 2010	rev 1.0
	original version
*)
END_FUNCTION_BLOCK

(* POU TN_RECEIVE, ST *)
FUNCTION_BLOCK TN_RECEIVE
VAR_IN_OUT
	R_BUF :	NETWORK_BUFFER;
	Xus_TN_SCREEN : us_TN_SCREEN;
END_VAR
VAR
	REQ_Size : UINT;
	REQ1 : BYTE;
	REQ2 : BYTE;
	REQ3 : BYTE;
END_VAR

(*
version 1.0		10. mai 2010
programmer		ks
tested by		ks

TN_RECEIVE empfängt Tastatureingaben vom Telnet Client und wertet diese aus
*)
(* Datenempfang auswertung *)
Xus_TN_SCREEN.by_Input_ASCII_Code := BYTE#00;
Xus_TN_SCREEN.by_Input_Exten_Code := BYTE#00;

IF R_BUF.SIZE > UINT#0 THEN
	(* empfangene Daten auswerten *)
	REQ_Size := R_BUF.SIZE;
	REQ1 := R_BUF.BUFFER[0];
	REQ2 := R_BUF.BUFFER[1];
	REQ3 := R_BUF.BUFFER[2];

	IF REQ1 = BYTE#27 AND REQ_Size >= UINT#3 THEN (* Escape *)
		IF REQ2 = BYTE#91 THEN (* Cursor code *)
			IF (REQ3 >= BYTE#65 AND REQ3 <= BYTE#68) OR (REQ3 = BYTE#72) OR (REQ3 = BYTE#75) THEN (* 65..68 = Cursor o,u,r,l / 72 = POS1 / 75 = ENDE *)
				Xus_TN_SCREEN.by_Input_Exten_Code := REQ3;
			END_IF;
		ELSIF REQ2 = BYTE#79 THEN (* Sondertasten F1/F2/F3/F4 *)
			IF REQ3 >= BYTE#80 AND REQ3 <= BYTE#83 THEN
				Xus_TN_SCREEN.by_Input_Exten_Code := REQ3;
			END_IF;
		END_IF;
	ELSIF REQ1 >= BYTE#32 AND REQ1 <= BYTE#126 THEN
		Xus_TN_SCREEN.by_Input_ASCII_Code := REQ1;
		Xus_TN_SCREEN.bo_Input_ASCII_IsNum := ISC_NUM(REQ1); (* Auswertung auf Zahleneingabe *)
	ELSIF REQ1 = BYTE#8 OR REQ1 = BYTE#9 OR REQ1 = BYTE#13 OR REQ1 = BYTE#27 THEN (* prüfe auf Steuerzeichen 8=Backspace / 9=Tabulator / 13=Return / 27=Escape *)
		Xus_TN_SCREEN.by_Input_Exten_Code := REQ1;
	END_IF;

	(* Empfangsbuffer Datenlänge null eintragen (Telegramm zerstören *)
	R_BUF.SIZE := UINT#00;
END_IF;

(* revision history
ks	10. mai. 2010	rev 1.0
	original version
*)
END_FUNCTION_BLOCK

(* POU TN_SEND_ROWS, ST *)
FUNCTION_BLOCK TN_SEND_ROWS
VAR_IN_OUT
	IP_C : IP_C;
	S_BUF : NETWORK_BUFFER;
	Xus_TN_SCREEN : us_TN_SCREEN;
END_VAR
VAR_INPUT
	S_BUF_SIZE : INT;
END_VAR
VAR
	in_Line_Count : INT;(*Zähler um max alle 24 Zeilen zu durchlaufen*)
	in_Col_Count : INT;
	in_Last_Row_Index : INT;
	bo_Break_Loop : BOOL;
	in_Row_Count : INT;
	in_Offset : INT;
	in_Write_Index : INT;
	in_Write_Index_Backup : INT;
	by_Cur_Color : BYTE;
	by_last_Color : BYTE;
	in_Write_Stop : INT;
END_VAR

(*
version 1.0		10. mai 2010
programmer		ks
tested by		ks

TN_SEND_ROWS prüft den Bildschirmspeicher auf änderungen, und sendet diese zeilenweise an den Telnet Client 
*)
(* Verbindung vorhanden und kein Datensenden aktiv *)
IF (IP_C.C_STATE < BYTE#127 OR S_BUF.SIZE > UINT#0) THEN
	RETURN; (* nein -> Baustein beenden *)
END_IF;

(* aktuellen Schreibindex laden *)
in_Write_Index := UINT_TO_INT(S_BUF.SIZE) - 1;

(* aktuellen Schreibindex zwischenspeichern *)
in_Write_Index_Backup := in_Write_Index;

(* positive Flanke Connect on *)
IF (IP_C.C_STATE = BYTE#254) OR (Xus_TN_SCREEN.bo_Clear_Screen) THEN

	(* Clear-Screen Meldung rücksetzen *)
	Xus_TN_SCREEN.bo_Clear_Screen := FALSE;

	(* alle Zeilen für Update markieren *)
	FOR in_Line_Count := INT#00 TO INT#23 DO
		Xus_TN_SCREEN.bya_Line_Update[in_Line_Count] := TRUE;
	END_FOR;

	(* ESC [0;30,40m  Reset Attributes + Black,Black *)
	in_Write_Index := in_Write_Index + INT#1;
	S_BUF.BUFFER[in_Write_Index] := BYTE#16#1B; (* ESC *)
	in_Write_Index := in_Write_Index + INT#1;
	S_BUF.BUFFER[in_Write_Index] := BYTE#16#5B; (* [ *)
	in_Write_Index := in_Write_Index + INT#1;
	S_BUF.BUFFER[in_Write_Index] := BYTE#16#30; (* 0 *)
	in_Write_Index := in_Write_Index + INT#1;
	S_BUF.BUFFER[in_Write_Index] := BYTE#16#3B; (* ; *)
	in_Write_Index := in_Write_Index + INT#1;
	S_BUF.BUFFER[in_Write_Index] := BYTE#16#33; (* 3 *)

	(* Einerstelle Farbe Foreground ausgeben *)
	in_Write_Index := in_Write_Index + INT#1;
	S_BUF.BUFFER[in_Write_Index] := (SHR(Xus_TN_SCREEN.by_Clear_Screen_Attr,4) OR BYTE#16#30);

	in_Write_Index := in_Write_Index + INT#1;
	S_BUF.BUFFER[in_Write_Index] := BYTE#16#3B; (* ; *)
	in_Write_Index := in_Write_Index + INT#1;
	S_BUF.BUFFER[in_Write_Index] := BYTE#16#34; (* 4 *)

	(* Einerstelle Farbe Background ausgeben *)
	in_Write_Index := in_Write_Index + INT#1;
	S_BUF.BUFFER[in_Write_Index] := ((Xus_TN_SCREEN.by_Clear_Screen_Attr AND BYTE#16#07) OR BYTE#16#30);

	in_Write_Index := in_Write_Index + INT#1;
	S_BUF.BUFFER[in_Write_Index] := BYTE#16#6D; (* m *)

	(* ESC[2J Clear screen and home cursor *)
	in_Write_Index := in_Write_Index + INT#1;
	S_BUF.BUFFER[in_Write_Index] := BYTE#16#1B; (* ESC *)
	in_Write_Index := in_Write_Index + INT#1;
	S_BUF.BUFFER[in_Write_Index] := BYTE#16#5B; (* [ *)
	in_Write_Index := in_Write_Index + INT#1;
	S_BUF.BUFFER[in_Write_Index] := BYTE#16#32; (* 2 *)
	in_Write_Index := in_Write_Index + INT#1;
	S_BUF.BUFFER[in_Write_Index] := BYTE#16#4A; (* J *)

	(* ESC [?7l Off *)
	in_Write_Index := in_Write_Index + INT#1;
	S_BUF.BUFFER[in_Write_Index] := BYTE#16#1B; (* ESC *)
	in_Write_Index := in_Write_Index + INT#1;
	S_BUF.BUFFER[in_Write_Index] := BYTE#16#5B; (* [ *)
	in_Write_Index := in_Write_Index + INT#1;
	S_BUF.BUFFER[in_Write_Index] := BYTE#16#3F; (* ? *)
	in_Write_Index := in_Write_Index + INT#1;
	S_BUF.BUFFER[in_Write_Index] := BYTE#16#37; (* 7 *)
	in_Write_Index := in_Write_Index + INT#1;
	S_BUF.BUFFER[in_Write_Index] := BYTE#16#6C; (* l *)

END_IF;

in_Last_Row_Index := INT#0;
bo_Break_Loop := FALSE;
in_Write_Stop := S_BUF_SIZE - 20;

(* alle Zeilen durchlaufen *)
FOR in_Line_Count := 0 TO 23 DO

	in_Offset := in_Row_Count * INT#80;

	(* prüfen ob Update einer Zeile notwendig ist bzw. nach Reconnect *)
	IF (Xus_TN_SCREEN.bya_Line_Update[in_Row_Count] = TRUE) THEN

		(* Schreib-Cursor positionieren *)
		in_Write_Index := in_Write_Index + INT#1;
		S_BUF.BUFFER[in_Write_Index] := BYTE#16#1B; (* ESC *)
		in_Write_Index := in_Write_Index + INT#1;
		S_BUF.BUFFER[in_Write_Index] := BYTE#16#5B; (* [ *)

		(* Zehnerstelle Zeilennummer ausgeben *)
		in_Write_Index := in_Write_Index + INT#1;
		S_BUF.BUFFER[in_Write_Index] :=
		SHR(INT_TO_BCDC(in_Row_Count + INT#1),INT#4) OR BYTE#16#30;

		(* Einerstelle Zeilennummer ausgeben *)
		in_Write_Index := in_Write_Index + INT#1;
		S_BUF.BUFFER[in_Write_Index] :=
		(INT_TO_BCDC(in_Row_Count + INT#1) AND BYTE#16#0F) OR BYTE#16#30;

		in_Write_Index := in_Write_Index + INT#1;
		S_BUF.BUFFER[in_Write_Index] := BYTE#16#3B; (* ; *)
		in_Write_Index := in_Write_Index + INT#1;
		S_BUF.BUFFER[in_Write_Index] := BYTE#16#31; (* 1 *)
		in_Write_Index := in_Write_Index + INT#1;
		S_BUF.BUFFER[in_Write_Index] := BYTE#16#48; (* H *)

		(* alle Spalten einer Zeile durchlaufen *)
		FOR in_Col_Count := 0 TO 79 DO

			(* aktuelle Farbe bestimmen *)
			by_Cur_Color := Xus_TN_SCREEN.bya_COLOR[in_Offset];
			IF (by_Cur_Color <> by_last_Color) OR (in_Col_Count = INT#00) THEN

				(* Farbeinstellung: ANSI-Sequenz ESC[X;Y;Zm ausgeben *)
				in_Write_Index := in_Write_Index + INT#1;
				S_BUF.BUFFER[in_Write_Index] := BYTE#16#1B; (* ESC *)

				in_Write_Index := in_Write_Index + INT#1;
				S_BUF.BUFFER[in_Write_Index] := BYTE#16#5B; (* [ *)

				(* Farbeinstellung: dunkel oder Hell und blinken bestimmen *)

					IF (((by_Cur_Color AND BYTE#2#10001000) XOR (by_last_Color AND BYTE#2#10001000)) <> BYTE#00) OR (in_Col_Count = 0) THEN

						in_Write_Index := in_Write_Index + INT#1;
						S_BUF.BUFFER[in_Write_Index] := BYTE#16#30; (* 0 *)
						in_Write_Index := in_Write_Index + INT#1;
						S_BUF.BUFFER[in_Write_Index] := BYTE#16#3B; (* ; *)

						(* keine dunklen Farben gewünscht -> dann Bold & Bright *)
						IF (by_Cur_Color AND BYTE#2#00001000) = BYTE#2#00000000 THEN

							(* auf Bold & Btight Farben umstellen *)
							in_Write_Index := in_Write_Index + INT#1;
							S_BUF.BUFFER[in_Write_Index] := BYTE#16#31; (* 1 *) 
							in_Write_Index := in_Write_Index + INT#1;
							S_BUF.BUFFER[in_Write_Index] := BYTE#16#3B; (* ; *)

						END_IF;

						(* blinkenden Farben gewünscht *)
						IF (by_Cur_Color AND BYTE#2#10000000) = BYTE#2#10000000 THEN 

							(* auf Bold & Bright Farben umstellen *)
							in_Write_Index := in_Write_Index + INT#1;
							S_BUF.BUFFER[in_Write_Index] := BYTE#16#35; (* 5 *) 
							in_Write_Index := in_Write_Index + INT#1;
							S_BUF.BUFFER[in_Write_Index] := BYTE#16#3B; (* ; *)

						END_IF;

					END_IF;

					(* Zehnerstelle Farbe Foreground ausgeben *)
					in_Write_Index := in_Write_Index + INT#1;
					S_BUF.BUFFER[in_Write_Index] := BYTE#16#33; (* 3 *)

					(* Einerstelle Farbe Foreground ausgeben *)
					in_Write_Index := in_Write_Index + INT#1;
					S_BUF.BUFFER[in_Write_Index] := ((SHR(by_Cur_Color,4) AND BYTE#2#00000111) OR BYTE#16#30);

					in_Write_Index := in_Write_Index + INT#1;
					S_BUF.BUFFER[in_Write_Index] := BYTE#16#3B; (* ; *)

					(* Zehnerstelle Farbe Background ausgeben *)
					in_Write_Index := in_Write_Index + INT#1;
					S_BUF.BUFFER[in_Write_Index] := BYTE#16#34; (* 4 *)

					(* Einerstelle Farbe Background ausgeben *)
					in_Write_Index := in_Write_Index + INT#1;
					S_BUF.BUFFER[in_Write_Index] := ((by_Cur_Color AND BYTE#2#00000111) OR BYTE#16#30); 

					in_Write_Index := in_Write_Index + INT#1;
					S_BUF.BUFFER[in_Write_Index] := BYTE#16#6D; (* m *)

					(* neue Farbe als letzt verwendete speichern *)
					by_last_Color := by_Cur_Color;

				END_IF;

				(* Buffer Ende vorzeitig erreicht -> Ende *)
				IF (in_Write_Index > in_Write_Stop) THEN

					bo_Break_Loop := TRUE;
					EXIT;

				END_IF;

				(* ein TEXT-Zeichen von Screenbuffer in den Sendebuffer übertragen *)
				in_Write_Index := in_Write_Index + INT#1;
				S_BUF.BUFFER[in_Write_Index] := Xus_TN_SCREEN.bya_CHAR[in_Offset];

				(* nächste Spalte anwählen *)
				in_Offset := in_Offset + INT#01;
			END_FOR;

			IF (bo_Break_Loop = TRUE) THEN;

				(* Buffer Ende vorzeitig erreicht -> nur bis zur letzten kompletten Zeile uebertragen *)
				in_Write_Index := in_Last_Row_Index;

				EXIT;
			END_IF;

			(* Buffer ist noch nicht voll -> neue Zeile ubernehmen *)
			in_Last_Row_Index := in_Write_Index;
			Xus_TN_SCREEN.bya_Line_Update[in_Row_Count] := FALSE;

		END_IF;

		(* naechste Zeile adressieren *)
		in_Row_Count := in_Row_Count + INT#01;

		(* ab letzter Zeile wieder von vorne beginnen *)
		IF (in_Row_Count > INT#23) THEN
			in_Row_Count := INT#00;
		END_IF;
		(*-----------------------------------------------*)


	END_FOR;

	(* wenn in einen Update-Zyklus alle Zeilen auf einmal geschafft wurden *)
	(* wird der Row_Count auf ersten Zeile gestellt *)
	(* soll das hässliche Grafikflackern verhindern *)
	(* ansonsten wird bei der letzen Zeile weitergemacht *)
	IF (bo_Break_Loop = FALSE) THEN
		in_Row_Count := INT#00;
	END_IF;

	(* Edit-Cursor positionieren *)
	IF (in_Write_Index <> in_Write_Index_Backup) THEN

		in_Write_Index := in_Write_Index + INT#1;
		S_BUF.BUFFER[in_Write_Index] := BYTE#16#1B; (* ESC *)
		in_Write_Index := in_Write_Index + INT#1;
		S_BUF.BUFFER[in_Write_Index] := BYTE#16#5B; (* [ *)

		(* Zehnerstelle Zeilennummer ausgeben *)
		in_Write_Index := in_Write_Index + INT#1;
		S_BUF.BUFFER[in_Write_Index] := SHR(INT_TO_BCDC(Xus_TN_SCREEN.in_Cursor_Y + 1),INT#4) OR BYTE#16#30;

		(* Einerstelle Zeilennummer ausgeben *)
		in_Write_Index := in_Write_Index + INT#1;
		S_BUF.BUFFER[in_Write_Index] := (INT_TO_BCDC(Xus_TN_SCREEN.in_Cursor_Y + 1) AND BYTE#16#0F) OR BYTE#16#30;

		in_Write_Index := in_Write_Index + INT#1;
		S_BUF.BUFFER[in_Write_Index] := BYTE#16#3B; (* ; *)

		(* Zehnerstelle Spaltenummer ausgeben *)
		in_Write_Index := in_Write_Index + INT#1;
		S_BUF.BUFFER[in_Write_Index] := SHR(INT_TO_BCDC(Xus_TN_SCREEN.in_Cursor_X + 1),INT#4) OR BYTE#16#30;

		(* Einerstelle Spaltennummer ausgeben *)
		in_Write_Index := in_Write_Index + INT#1;
		S_BUF.BUFFER[in_Write_Index] := (INT_TO_BCDC(Xus_TN_SCREEN.in_Cursor_X + 1) AND BYTE#16#0F) OR BYTE#16#30;

		in_Write_Index := in_Write_Index + INT#1;
		S_BUF.BUFFER[in_Write_Index] := BYTE#16#48; (* H *)

END_IF;

(* aktuellen Schreibindex speichern -> Senden anstossen *)
S_BUF.SIZE := INT_TO_UINT(in_Write_Index + 1);

(* revision history
ks	10. mai. 2010	rev 1.0
	original version
*)
END_FUNCTION_BLOCK

(* POU LOG_VIEWPORT, ST *)
FUNCTION_BLOCK LOG_VIEWPORT
VAR_IN_OUT
	LC : LOG_CONTROL;
	LV : us_LOG_VIEWPORT;
END_VAR
VAR
	pos : INT;
	count : INT;
	idx : INT;
	base : INT;
	update_pos : BOOL;
END_VAR

(*
version 1.1		05 mai 2012
programmer		ks
tested BY		ks

LOG_VIEWPORT erzeugt einen Liste der Meldungen des Loggingbuffers die innerhalb einer virtuellen Ansicht enthalten sind.
*)
(* Scroll Button verarbeiten *)
IF LV.MOVE_TO_X <> 0 THEN
	CASE LV.MOVE_TO_X OF
	30000: pos := 1 ; (* älteste Meldung anzeigen *)
	30001: pos := LC.SIZE; (* neueste Meldung anzeigen *)
	30002: pos := pos + LV.COUNT; (* eine Seite nach unten blättern -> Richtung neuere Nachrichten *)
	30003: pos := pos - LV.COUNT; (* eine Seite nach oben blättern -> Richtung ältere Nachrichten *)
	ELSE
		pos := pos + LV.MOVE_TO_X;
	END_CASE;
	update_pos := TRUE;
	LV.MOVE_TO_X := 0;
END_IF;

IF (LV.UPDATE_COUNT <> LC.UPDATE_COUNT) OR update_pos THEN (* Aktualisierung überwachen *)
	LV.UPDATE := TRUE;
	LV.UPDATE_COUNT := LC.UPDATE_COUNT;
	update_pos := FALSE;

	(* pos prüfen und übernehmen *)
	IF LC.RING_MODE THEN
		pos := LIMIT(1,pos,LC.SIZE - LV.COUNT + 1);
	ELSE
		IF LC.IDX > LV.COUNT THEN
			pos := LIMIT(1,pos,LC.IDX - LV.COUNT + 1);
		ELSE
			pos := 1;
		END_IF;
	END_IF;

	(* idxBasis berechnen *)
	base := LC.IDX - pos - LV.COUNT + 1;
	IF LC.RING_MODE THEN 
		(* Anzeige im Ringpuffermodus *)
		FOR count:= 1 TO LV.COUNT DO
			idx := base + count;
			IF idx < 1 THEN
				idx := idx + LC.SIZE;
			END_IF;
			LV.LINE_ARRAY[count] := idx;
		END_FOR;
	ELSE
		(* Anzeige im Normalmodus *)
		FOR count:= 1 TO LV.COUNT DO
			idx := base + count;
			IF idx < 1 THEN
				(* Leere Zeile ausgeben *)
				LV.LINE_ARRAY[count] := 0;
			ELSE
				LV.LINE_ARRAY[count] := idx;
			END_IF;
		END_FOR;
	END_IF;
END_IF;

(* revision history
ks	01. mai 2010	rev 1.0
	original version

ks	05. mai 2012	rev 1.1
	Fehler im Ringmodus

*)
END_FUNCTION_BLOCK

(* POU TN_SC_VIEWPORT, ST *)
FUNCTION_BLOCK TN_SC_VIEWPORT
VAR
	FB_TN_SC_WRITE : TN_SC_WRITE;
	FB_TON : TON;
END_VAR
VAR
	in_index : INT;
	in_Color : INT;
	by_Attr : BYTE;
	in_count : INT;
END_VAR
VAR_IN_OUT
	Xus_LOG_VIEWPORT : us_LOG_VIEWPORT;
	Xus_LOG_CONTROL : LOG_CONTROL;
	Xus_TN_SCREEN : us_TN_SCREEN;
END_VAR
VAR_INPUT
	Iin_X : INT;
	Iin_Y : INT;
	Iin_Width : INT;
	Idw_ATTR_1 : DWORD;
	Idw_ATTR_2 : DWORD;
	Iti_TIME : TIME;
END_VAR

(*
version 1.0		10. mai 2010
programmer		ks
tested by		ks

TN_SC_VIEWPORT verwaltet und zeichnet einen rechteckigen Bereich in dem der Log-buffer angezeigt wird
*)
(* LOG-Messages ausgeben *)

IF Xus_LOG_VIEWPORT.UPDATE AND FB_TON.Q THEN (* Update gewünscht und Verzögerungszeit abgelaufen *)
	Xus_LOG_VIEWPORT.UPDATE := FALSE;
	FOR in_count := 1 TO Xus_LOG_VIEWPORT.COUNT DO (* Alle Viewport-Zeilen abarbeiten *)
		in_index := Xus_LOG_VIEWPORT.LINE_ARRAY[in_count];
		(* Farbe aus den Option-Parameter auslesen >0,Level,Back,Front< *)
		in_Color := DWORD_TO_INT(Xus_LOG_CONTROL.MSG_OPTION[in_index] AND DWORD#2#1111);

		CASE in_Color OF
		0..3: by_Attr := BYTE_OF_DWORD(Idw_ATTR_1,INT_TO_BYTE(in_Color));
		4..7: by_Attr := BYTE_OF_DWORD(Idw_ATTR_2,INT_TO_BYTE(in_Color));
		ELSE
			by_Attr := BYTE_OF_DWORD(Idw_ATTR_1,BYTE#0);
		END_CASE;

		(* Message (Text + Farbe) ausgeben *)
		FB_TN_SC_WRITE(	Iin_Y := Iin_Y + in_count - INT#01,
						Iin_X := Iin_X,
						Iby_ATTR := by_Attr,
						Ist_STRING := FIX(str := Xus_LOG_CONTROL.MSG[in_index], L := Iin_Width, C := BYTE#32, M := INT#00), (* String rechts ergänzen bzw. kürzen *)
						Xus_TN_SCREEN := Xus_TN_SCREEN);

	END_FOR;

	(* Timer stoppen/rücksetzen *)
	FB_TON.IN := FALSE;
	FB_TON.PT := Iti_TIME;
	FB_TON();

END_IF;

(* Update-Zeitverzoegerung *)
FB_TON.IN := TRUE;
FB_TON.PT := Iti_TIME;
FB_TON();

(* revision history
ks	10. mai. 2010	rev 1.0
	original version
*)
END_FUNCTION_BLOCK

(* POU TN_VISION_DEMO_2, ST *)
PROGRAM TN_VISION_DEMO_2
VAR
	FB_TN_FRAMEWORK : TN_FRAMEWORK;
	FB_TN_SC_FILL : TN_SC_FILL;
	FB_TN_SC_WRITE_C : TN_SC_WRITE_C;
	FB_TN_SC_WRITE : TN_SC_WRITE;
	Xus_TN_MENU : us_TN_MENU;
	Xus_TN_INPUT_CONTROL : us_TN_INPUT_CONTROL;
	Xus_TN_SCREEN : us_TN_SCREEN;
	S_BUF : NETWORK_BUFFER;
	R_BUF : NETWORK_BUFFER;
	IP_C : IP_C;
END_VAR
FB_TN_FRAMEWORK(
					us_TN_INPUT_CONTROL := Xus_TN_INPUT_CONTROL ,
					us_TN_SCREEN := Xus_TN_SCREEN ,
					us_TN_MENU := Xus_TN_MENU ,
					S_BUF := S_BUF ,
					R_BUF:= R_BUF ,
					IP_C:= IP_C ,
					PORT := WORD#0
					 );


(* Initialisierung der Daten und Strukturen *)
IF (Xus_TN_SCREEN.in_Page_Number = INT#00) THEN
	Xus_TN_SCREEN.in_Page_Number := INT#01;

	(* Clear-Screen (Farbe setzen + Display löschen) *)
	Xus_TN_SCREEN.by_Clear_Screen_Attr := BYTE#16#00;
	Xus_TN_SCREEN.bo_Clear_Screen := TRUE;

	(* Screen initialisieren (mit Leerzeichen füllen) *)
	FB_TN_SC_FILL(	Iin_X1 := INT#00,
					Iin_Y1 := INT#00,
					Iin_X2 := INT#79,
					Iin_Y2 := INT#23,
					Iby_CHAR := BYTE#32,
					Iby_Attr := BYTE#16#00,
					Xus_TN_SCREEN := Xus_TN_SCREEN);

	(* Statische Texte ausgeben *)
	FB_TN_SC_WRITE(	Iin_X := INT#00,
					Iin_Y := INT#00,
					Iby_ATTR := BYTE#16#70,
					Ist_STRING := 'Login Screen                                                     FL SWITCH MM HS',
					Xus_TN_SCREEN := Xus_TN_SCREEN);

	(* Statische Texte ausgeben *)
	FB_TN_SC_WRITE(	Iin_X := INT#00,
					Iin_Y := INT#03,
					Iby_ATTR := BYTE#16#70,
					Ist_STRING := 'XXXXXXXXX',
					Xus_TN_SCREEN := Xus_TN_SCREEN);

	(* Statische Texte ausgeben *)
	FB_TN_SC_WRITE(	Iin_X := INT#00,
					Iin_Y := INT#04,
					Iby_ATTR := BYTE#16#70,
					Ist_STRING := 'X   X  XX',
					Xus_TN_SCREEN := Xus_TN_SCREEN);

	(* Statische Texte ausgeben *)
	FB_TN_SC_WRITE(	Iin_X := INT#00,
					Iin_Y := INT#05,
					Iby_ATTR := BYTE#16#70,
					Ist_STRING := 'X   O   X      ---> Phoenix Contact Managed Switch System <---',
					Xus_TN_SCREEN := Xus_TN_SCREEN);

	(* Statische Texte ausgeben *)
	FB_TN_SC_WRITE(	Iin_X := INT#00,
					Iin_Y := INT#06,
					Iby_ATTR := BYTE#16#70,
					Ist_STRING := 'X   X  XX               Phoenix Contact GmbH & Co KG',
					Xus_TN_SCREEN := Xus_TN_SCREEN);

	(* Statische Texte ausgeben *)
	FB_TN_SC_WRITE(	Iin_X := INT#00,
					Iin_Y := INT#07,
					Iby_ATTR := BYTE#16#70,
					Ist_STRING := 'X   XXXXX                   www.PhoenixContact.com',
					Xus_TN_SCREEN := Xus_TN_SCREEN);

	(* Statische Texte ausgeben *)
	FB_TN_SC_WRITE(	Iin_X := INT#00,
					Iin_Y := INT#08,
					Iby_ATTR := BYTE#16#70,
					Ist_STRING := 'X   XXXXX',
					Xus_TN_SCREEN := Xus_TN_SCREEN);

	(* Statische Texte ausgeben *)
	FB_TN_SC_WRITE(	Iin_X := INT#00,
					Iin_Y := INT#09,
					Iby_ATTR := BYTE#16#70,
					Ist_STRING := 'XXXXXXXXX',
					Xus_TN_SCREEN := Xus_TN_SCREEN);

	(* Statische Texte ausgeben *)
	FB_TN_SC_WRITE(	Iin_X := INT#00,
					Iin_Y := INT#11,
					Iby_ATTR := BYTE#16#70,
					Ist_STRING := '                Running switch application version:  4.00',
					Xus_TN_SCREEN := Xus_TN_SCREEN);

	(* Alle Input-Controls initialisieren *)

	Xus_TN_INPUT_CONTROL.bo_Enable := FALSE;

  (* Initialisierung der Eingabe-Zeile *)
	Xus_TN_INPUT_CONTROL.usa_TN_INPUT_CONTROL_DATA[1].in_Type := INT#01;
	Xus_TN_INPUT_CONTROL.usa_TN_INPUT_CONTROL_DATA[1].in_Y := INT#17;
	Xus_TN_INPUT_CONTROL.usa_TN_INPUT_CONTROL_DATA[1].in_X := INT#33;
	Xus_TN_INPUT_CONTROL.usa_TN_INPUT_CONTROL_DATA[1].by_Attr_mF := BYTE#16#70;
	Xus_TN_INPUT_CONTROL.usa_TN_INPUT_CONTROL_DATA[1].by_Attr_oF := BYTE#16#70;
	Xus_TN_INPUT_CONTROL.usa_TN_INPUT_CONTROL_DATA[1].in_Cursor_Pos := INT#0;
	Xus_TN_INPUT_CONTROL.usa_TN_INPUT_CONTROL_DATA[1].bo_Input_Only_Num := FALSE;
	Xus_TN_INPUT_CONTROL.usa_TN_INPUT_CONTROL_DATA[1].bo_Input_Hidden := TRUE;
	Xus_TN_INPUT_CONTROL.usa_TN_INPUT_CONTROL_DATA[1].st_Input_Mask := '                ';
	Xus_TN_INPUT_CONTROL.usa_TN_INPUT_CONTROL_DATA[1].st_Input_Data := Xus_TN_INPUT_CONTROL.usa_TN_INPUT_CONTROL_DATA[1].st_Input_Mask;
	Xus_TN_INPUT_CONTROL.usa_TN_INPUT_CONTROL_DATA[1].st_Input_ToolTip := '';
	Xus_TN_INPUT_CONTROL.usa_TN_INPUT_CONTROL_DATA[1].in_Input_Option := INT#00;
	Xus_TN_INPUT_CONTROL.usa_TN_INPUT_CONTROL_DATA[1].in_Title_Y_Offset := INT#00;
	Xus_TN_INPUT_CONTROL.usa_TN_INPUT_CONTROL_DATA[1].in_Title_X_Offset := -12;
	Xus_TN_INPUT_CONTROL.usa_TN_INPUT_CONTROL_DATA[1].by_Title_Attr := BYTE#16#70;
	Xus_TN_INPUT_CONTROL.usa_TN_INPUT_CONTROL_DATA[1].st_Title_String := 'Password:  [                ]';

	(* Control-Tool-Tip *)
	Xus_TN_INPUT_CONTROL.in_ToolTip_Y := INT#23;
	Xus_TN_INPUT_CONTROL.in_ToolTip_X := INT#09;
	Xus_TN_INPUT_CONTROL.by_ToolTip_Attr := BYTE#16#70;
	Xus_TN_INPUT_CONTROL.in_ToolTip_Size := INT#30;

	(* Control-Verwaltung initialisieren *)
	Xus_TN_INPUT_CONTROL.in_Count := INT#01;
	Xus_TN_INPUT_CONTROL.bo_Enable := TRUE;
	Xus_TN_INPUT_CONTROL.bo_Reset_Fokus := TRUE;
END_IF;

IF (Xus_TN_SCREEN.in_Page_Number = INT#01) THEN

	(* eingegebenen String übernehmen *)
	IF Xus_TN_INPUT_CONTROL.usa_TN_INPUT_CONTROL_DATA[1].bo_Input_Entered = TRUE THEN

		Xus_TN_INPUT_CONTROL.usa_TN_INPUT_CONTROL_DATA[1].bo_Input_Entered := FALSE;

		Xus_TN_INPUT_CONTROL.usa_TN_INPUT_CONTROL_DATA[1].st_Input_String :=
			LOWERCASE(str:=Xus_TN_INPUT_CONTROL.usa_TN_INPUT_CONTROL_DATA[1].st_Input_String);

		IF Xus_TN_INPUT_CONTROL.usa_TN_INPUT_CONTROL_DATA[1].st_Input_String = 'oscat' THEN
			Xus_TN_SCREEN.in_Page_Number := INT#04;

		ELSE
			FB_TN_SC_WRITE_C(	Iin_Y := Xus_TN_INPUT_CONTROL.in_ToolTip_Y,
								Iin_X := Xus_TN_INPUT_CONTROL.in_ToolTip_X,
								Iby_ATTR := BYTE#16#F1,
								Iin_OPTION := INT#02, (* Center-String *)
								Iin_LENGTH := Xus_TN_INPUT_CONTROL.in_ToolTip_Size,
								Ist_STRING := ' User Password Failed   ',
								Xus_TN_SCREEN := Xus_TN_SCREEN);
		END_IF;
	END_IF;
END_IF;

(* Initialisierung der Daten und Strukturen *)
IF (Xus_TN_SCREEN.in_Page_Number = INT#04) THEN
	Xus_TN_SCREEN.in_Page_Number := INT#05;

	(* Clear-Screen (Farbe setzen + Display löschen) *)
	Xus_TN_SCREEN.by_Clear_Screen_Attr := BYTE#16#00;
	Xus_TN_SCREEN.bo_Clear_Screen := TRUE;

	(* Screen initialisieren (mit Leerzeichen füllen) *)
	FB_TN_SC_FILL(	Iin_X1 := INT#00,
					Iin_Y1 := INT#00,
					Iin_X2 := INT#79,
					Iin_Y2 := INT#23,
					Iby_CHAR := BYTE#32,
					Iby_Attr := BYTE#16#00,
					Xus_TN_SCREEN := Xus_TN_SCREEN);

	(* Statische Texte ausgeben *)
	FB_TN_SC_WRITE(	Iin_X := INT#00,
					Iin_Y := INT#00,
					Iby_ATTR := BYTE#16#70,
					Ist_STRING := 'Basic Switch Configuration                                       FL SWITCH MM HS',
					Xus_TN_SCREEN := Xus_TN_SCREEN);

	(* Statische Texte ausgeben                                         *)
	FB_TN_SC_WRITE(	Iin_X := INT#00,
					Iin_Y := INT#03,
					Iby_ATTR := BYTE#16#70,
					Ist_STRING := 'XXXXXXXXX        MAC Address             : 00:A0:45:00:6E:9B',
					Xus_TN_SCREEN := Xus_TN_SCREEN);

	(* Statische Texte ausgeben *)
	FB_TN_SC_WRITE(	Iin_X := INT#00,
					Iin_Y := INT#04,
					Iby_ATTR := BYTE#16#70,
					Ist_STRING := 'X   X  XX',
					Xus_TN_SCREEN := Xus_TN_SCREEN);

	(* Statische Texte ausgeben *)
	FB_TN_SC_WRITE(	Iin_X := INT#00,
					Iin_Y := INT#05,
					Iby_ATTR := BYTE#16#70,
					Ist_STRING := 'X   O   X',
					Xus_TN_SCREEN := Xus_TN_SCREEN);

	(* Statische Texte ausgeben *)
	FB_TN_SC_WRITE(	Iin_X := INT#00,
					Iin_Y := INT#06,
					Iby_ATTR := BYTE#16#70,
					Ist_STRING := 'X   X  XX',
					Xus_TN_SCREEN := Xus_TN_SCREEN);

	(* Statische Texte ausgeben *)
	FB_TN_SC_WRITE(	Iin_X := INT#00,
					Iin_Y := INT#07,
					Iby_ATTR := BYTE#16#70,
					Ist_STRING := 'X   XXXXX',
					Xus_TN_SCREEN := Xus_TN_SCREEN);

	(* Statische Texte ausgeben *)
	FB_TN_SC_WRITE(	Iin_X := INT#00,
					Iin_Y := INT#08,
					Iby_ATTR := BYTE#16#70,
					Ist_STRING := 'X   XXXXX',
					Xus_TN_SCREEN := Xus_TN_SCREEN);

	(* Statische Texte ausgeben *)
	FB_TN_SC_WRITE(	Iin_X := INT#00,
					Iin_Y := INT#09,
					Iby_ATTR := BYTE#16#70,
					Ist_STRING := 'XXXXXXXXX',
					Xus_TN_SCREEN := Xus_TN_SCREEN);

	(* Alle Input-Controls initialisieren *)

	Xus_TN_INPUT_CONTROL.bo_Enable      := FALSE;

	Xus_TN_INPUT_CONTROL.usa_TN_INPUT_CONTROL_DATA[1].in_Type := INT#01;
	Xus_TN_INPUT_CONTROL.usa_TN_INPUT_CONTROL_DATA[1].in_Y := INT#04;
	Xus_TN_INPUT_CONTROL.usa_TN_INPUT_CONTROL_DATA[1].in_X := INT#44;
	Xus_TN_INPUT_CONTROL.usa_TN_INPUT_CONTROL_DATA[1].by_Attr_mF := BYTE#16#07; (* Weiss, Grün *)
	Xus_TN_INPUT_CONTROL.usa_TN_INPUT_CONTROL_DATA[1].by_Attr_oF := BYTE#16#70; (* Weiss, Blau *)
	Xus_TN_INPUT_CONTROL.usa_TN_INPUT_CONTROL_DATA[1].in_Cursor_Pos := INT#0;
	Xus_TN_INPUT_CONTROL.usa_TN_INPUT_CONTROL_DATA[1].bo_Input_Only_Num := TRUE;
	Xus_TN_INPUT_CONTROL.usa_TN_INPUT_CONTROL_DATA[1].bo_Input_Hidden := FALSE;
	Xus_TN_INPUT_CONTROL.usa_TN_INPUT_CONTROL_DATA[1].st_Input_Mask := '   .   .   .   ';
	Xus_TN_INPUT_CONTROL.usa_TN_INPUT_CONTROL_DATA[1].st_Input_Data := Xus_TN_INPUT_CONTROL.usa_TN_INPUT_CONTROL_DATA[1].st_Input_Mask;
	Xus_TN_INPUT_CONTROL.usa_TN_INPUT_CONTROL_DATA[1].st_Input_ToolTip := 'Enter Agent IP Address in decimal dot format (e.g., 209.131.209.13)';
	Xus_TN_INPUT_CONTROL.usa_TN_INPUT_CONTROL_DATA[1].in_Input_Option := INT#01;
	Xus_TN_INPUT_CONTROL.usa_TN_INPUT_CONTROL_DATA[1].in_Title_Y_Offset := INT#00;
	Xus_TN_INPUT_CONTROL.usa_TN_INPUT_CONTROL_DATA[1].in_Title_X_Offset := -27;
	Xus_TN_INPUT_CONTROL.usa_TN_INPUT_CONTROL_DATA[1].by_Title_Attr := BYTE#16#70;
	Xus_TN_INPUT_CONTROL.usa_TN_INPUT_CONTROL_DATA[1].st_Title_String := 'IP Address              : [149.208.100.100]';

	Xus_TN_INPUT_CONTROL.usa_TN_INPUT_CONTROL_DATA[2].in_Type := INT#01;
	Xus_TN_INPUT_CONTROL.usa_TN_INPUT_CONTROL_DATA[2].in_Y := INT#05;
	Xus_TN_INPUT_CONTROL.usa_TN_INPUT_CONTROL_DATA[2].in_X := INT#44;
	Xus_TN_INPUT_CONTROL.usa_TN_INPUT_CONTROL_DATA[2].by_Attr_mF := BYTE#16#07; (* Weiss, Grün *)
	Xus_TN_INPUT_CONTROL.usa_TN_INPUT_CONTROL_DATA[2].by_Attr_oF := BYTE#16#70; (* Weiss, Blau *)
	Xus_TN_INPUT_CONTROL.usa_TN_INPUT_CONTROL_DATA[2].in_Cursor_Pos := INT#0;
	Xus_TN_INPUT_CONTROL.usa_TN_INPUT_CONTROL_DATA[2].bo_Input_Only_Num := TRUE;
	Xus_TN_INPUT_CONTROL.usa_TN_INPUT_CONTROL_DATA[2].bo_Input_Hidden := FALSE;
	Xus_TN_INPUT_CONTROL.usa_TN_INPUT_CONTROL_DATA[2].st_Input_Mask := '   .   .   .   ';
	Xus_TN_INPUT_CONTROL.usa_TN_INPUT_CONTROL_DATA[2].st_Input_Data := Xus_TN_INPUT_CONTROL.usa_TN_INPUT_CONTROL_DATA[1].st_Input_Mask;
	Xus_TN_INPUT_CONTROL.usa_TN_INPUT_CONTROL_DATA[2].st_Input_ToolTip := 'Enter Agent Netmask (e.g., 255.255.255.0)';
	Xus_TN_INPUT_CONTROL.usa_TN_INPUT_CONTROL_DATA[2].in_Input_Option := INT#01;
	Xus_TN_INPUT_CONTROL.usa_TN_INPUT_CONTROL_DATA[2].in_Title_Y_Offset := INT#00;
	Xus_TN_INPUT_CONTROL.usa_TN_INPUT_CONTROL_DATA[2].in_Title_X_Offset := -27;
	Xus_TN_INPUT_CONTROL.usa_TN_INPUT_CONTROL_DATA[2].by_Title_Attr := BYTE#16#70;
	Xus_TN_INPUT_CONTROL.usa_TN_INPUT_CONTROL_DATA[2].st_Title_String := 'Subnet Mask             : [255.255.255.128]';

	Xus_TN_INPUT_CONTROL.usa_TN_INPUT_CONTROL_DATA[3].in_Type := INT#01;
	Xus_TN_INPUT_CONTROL.usa_TN_INPUT_CONTROL_DATA[3].in_Y := INT#06;
	Xus_TN_INPUT_CONTROL.usa_TN_INPUT_CONTROL_DATA[3].in_X := INT#44;
	Xus_TN_INPUT_CONTROL.usa_TN_INPUT_CONTROL_DATA[3].by_Attr_mF := BYTE#16#07; (* Weiss, Grün *)
	Xus_TN_INPUT_CONTROL.usa_TN_INPUT_CONTROL_DATA[3].by_Attr_oF := BYTE#16#70; (* Weiss, Blau *)
	Xus_TN_INPUT_CONTROL.usa_TN_INPUT_CONTROL_DATA[3].in_Cursor_Pos := INT#0;
	Xus_TN_INPUT_CONTROL.usa_TN_INPUT_CONTROL_DATA[3].bo_Input_Only_Num := TRUE;
	Xus_TN_INPUT_CONTROL.usa_TN_INPUT_CONTROL_DATA[3].bo_Input_Hidden := FALSE;
	Xus_TN_INPUT_CONTROL.usa_TN_INPUT_CONTROL_DATA[3].st_Input_Mask := '   .   .   .   ';
	Xus_TN_INPUT_CONTROL.usa_TN_INPUT_CONTROL_DATA[3].st_Input_Data := Xus_TN_INPUT_CONTROL.usa_TN_INPUT_CONTROL_DATA[1].st_Input_Mask;
	Xus_TN_INPUT_CONTROL.usa_TN_INPUT_CONTROL_DATA[3].st_Input_ToolTip := 'Enter Agent Default Gateway, (e.g., 209.131.209.1)';
	Xus_TN_INPUT_CONTROL.usa_TN_INPUT_CONTROL_DATA[3].in_Input_Option := INT#01;
	Xus_TN_INPUT_CONTROL.usa_TN_INPUT_CONTROL_DATA[3].in_Title_Y_Offset := INT#00;
	Xus_TN_INPUT_CONTROL.usa_TN_INPUT_CONTROL_DATA[3].in_Title_X_Offset := -27;
	Xus_TN_INPUT_CONTROL.usa_TN_INPUT_CONTROL_DATA[3].by_Title_Attr := BYTE#16#70;
	Xus_TN_INPUT_CONTROL.usa_TN_INPUT_CONTROL_DATA[3].st_Title_String := 'Default Gateway         : [149.208.100.1  ]';

	Xus_TN_INPUT_CONTROL.usa_TN_INPUT_CONTROL_DATA[4].in_Type := INT#02;
	Xus_TN_INPUT_CONTROL.usa_TN_INPUT_CONTROL_DATA[4].in_Y := INT#07;
	Xus_TN_INPUT_CONTROL.usa_TN_INPUT_CONTROL_DATA[4].in_X := INT#44;
	Xus_TN_INPUT_CONTROL.usa_TN_INPUT_CONTROL_DATA[4].by_Attr_mF := BYTE#16#07;
	Xus_TN_INPUT_CONTROL.usa_TN_INPUT_CONTROL_DATA[4].by_Attr_oF := BYTE#16#70;
	Xus_TN_INPUT_CONTROL.usa_TN_INPUT_CONTROL_DATA[4].st_Input_Mask := '       ';
	Xus_TN_INPUT_CONTROL.usa_TN_INPUT_CONTROL_DATA[4].st_Input_Data := 'BootP  #DHCP   #DCP    #Static ';
	Xus_TN_INPUT_CONTROL.usa_TN_INPUT_CONTROL_DATA[4].st_Input_ToolTip := 'Push SPACE to select the address assignment (effective after reboot)';
	Xus_TN_INPUT_CONTROL.usa_TN_INPUT_CONTROL_DATA[4].in_Input_Option := INT#02;
	Xus_TN_INPUT_CONTROL.usa_TN_INPUT_CONTROL_DATA[4].in_Title_Y_Offset := INT#00;
	Xus_TN_INPUT_CONTROL.usa_TN_INPUT_CONTROL_DATA[4].in_Title_X_Offset := -27;
	Xus_TN_INPUT_CONTROL.usa_TN_INPUT_CONTROL_DATA[4].by_Title_Attr := BYTE#16#70;
	Xus_TN_INPUT_CONTROL.usa_TN_INPUT_CONTROL_DATA[4].st_Title_String := 'IP Parameter Assignment : <BootP  >';

	Xus_TN_INPUT_CONTROL.usa_TN_INPUT_CONTROL_DATA[5].in_Type := INT#02;
	Xus_TN_INPUT_CONTROL.usa_TN_INPUT_CONTROL_DATA[5].in_Y := INT#09;
	Xus_TN_INPUT_CONTROL.usa_TN_INPUT_CONTROL_DATA[5].in_X := INT#44;
	Xus_TN_INPUT_CONTROL.usa_TN_INPUT_CONTROL_DATA[5].by_Attr_mF := BYTE#16#07;
	Xus_TN_INPUT_CONTROL.usa_TN_INPUT_CONTROL_DATA[5].by_Attr_oF := BYTE#16#70;
	Xus_TN_INPUT_CONTROL.usa_TN_INPUT_CONTROL_DATA[5].st_Input_Mask := '                              ';
	Xus_TN_INPUT_CONTROL.usa_TN_INPUT_CONTROL_DATA[5].st_Input_Data := 'No Redundancy#Rapid Spanning Tree, Disabled#Rapid Spanning Tree, Enabled';
	Xus_TN_INPUT_CONTROL.usa_TN_INPUT_CONTROL_DATA[5].st_Input_ToolTip := 'Push SPACE to chose redundancy (network disruption for few seconds if enabled)';
	Xus_TN_INPUT_CONTROL.usa_TN_INPUT_CONTROL_DATA[5].in_Input_Option := INT#02;
	Xus_TN_INPUT_CONTROL.usa_TN_INPUT_CONTROL_DATA[5].in_Title_Y_Offset := INT#00;
	Xus_TN_INPUT_CONTROL.usa_TN_INPUT_CONTROL_DATA[5].in_Title_X_Offset := -27;
	Xus_TN_INPUT_CONTROL.usa_TN_INPUT_CONTROL_DATA[5].by_Title_Attr := BYTE#16#70;
	Xus_TN_INPUT_CONTROL.usa_TN_INPUT_CONTROL_DATA[5].st_Title_String := 'Redundancy              : <No Redundancy                 >';

	(* Statische Texte ausgeben *)
	FB_TN_SC_WRITE(	Iin_X := INT#17,
					Iin_Y := INT#10,
					Iby_ATTR := BYTE#16#70,
					Ist_STRING := 'Current Vlan Status     :  VLAN Transparent',
					Xus_TN_SCREEN := Xus_TN_SCREEN);

	Xus_TN_INPUT_CONTROL.usa_TN_INPUT_CONTROL_DATA[6].in_Type := INT#02;
	Xus_TN_INPUT_CONTROL.usa_TN_INPUT_CONTROL_DATA[6].in_Y := INT#11;
	Xus_TN_INPUT_CONTROL.usa_TN_INPUT_CONTROL_DATA[6].in_X := INT#44;
	Xus_TN_INPUT_CONTROL.usa_TN_INPUT_CONTROL_DATA[6].by_Attr_mF := BYTE#16#07;
	Xus_TN_INPUT_CONTROL.usa_TN_INPUT_CONTROL_DATA[6].by_Attr_oF := BYTE#16#70;
	Xus_TN_INPUT_CONTROL.usa_TN_INPUT_CONTROL_DATA[6].st_Input_Mask := '                        ';
	Xus_TN_INPUT_CONTROL.usa_TN_INPUT_CONTROL_DATA[6].st_Input_Data := 'VLAN Transparent#VLAN Tagging';
	Xus_TN_INPUT_CONTROL.usa_TN_INPUT_CONTROL_DATA[6].st_Input_ToolTip := 'Push SPACE to toggle the VLAN Mode (effective after reboot)';
	Xus_TN_INPUT_CONTROL.usa_TN_INPUT_CONTROL_DATA[6].in_Input_Option := INT#02;
	Xus_TN_INPUT_CONTROL.usa_TN_INPUT_CONTROL_DATA[6].in_Title_Y_Offset := INT#00;
	Xus_TN_INPUT_CONTROL.usa_TN_INPUT_CONTROL_DATA[6].in_Title_X_Offset := -27;
	Xus_TN_INPUT_CONTROL.usa_TN_INPUT_CONTROL_DATA[6].by_Title_Attr := BYTE#16#70;
	Xus_TN_INPUT_CONTROL.usa_TN_INPUT_CONTROL_DATA[6].st_Title_String := 'Vlan Mode               : <VLAN Transparent        >';

	Xus_TN_INPUT_CONTROL.usa_TN_INPUT_CONTROL_DATA[7].in_Type := INT#02;
	Xus_TN_INPUT_CONTROL.usa_TN_INPUT_CONTROL_DATA[7].in_Y := INT#12;
	Xus_TN_INPUT_CONTROL.usa_TN_INPUT_CONTROL_DATA[7].in_X := INT#44;
	Xus_TN_INPUT_CONTROL.usa_TN_INPUT_CONTROL_DATA[7].by_Attr_mF := BYTE#16#07;
	Xus_TN_INPUT_CONTROL.usa_TN_INPUT_CONTROL_DATA[7].by_Attr_oF := BYTE#16#70;
	Xus_TN_INPUT_CONTROL.usa_TN_INPUT_CONTROL_DATA[7].st_Input_Mask := '       ';
	Xus_TN_INPUT_CONTROL.usa_TN_INPUT_CONTROL_DATA[7].st_Input_Data := 'Disable#Enable';
	Xus_TN_INPUT_CONTROL.usa_TN_INPUT_CONTROL_DATA[7].st_Input_ToolTip := 'Push SPACE to Enable/Disable Port Security';
	Xus_TN_INPUT_CONTROL.usa_TN_INPUT_CONTROL_DATA[7].in_Input_Option := INT#02;
	Xus_TN_INPUT_CONTROL.usa_TN_INPUT_CONTROL_DATA[7].in_Title_Y_Offset := INT#00;
	Xus_TN_INPUT_CONTROL.usa_TN_INPUT_CONTROL_DATA[7].in_Title_X_Offset := -27;
	Xus_TN_INPUT_CONTROL.usa_TN_INPUT_CONTROL_DATA[7].by_Title_Attr := BYTE#16#70;
	Xus_TN_INPUT_CONTROL.usa_TN_INPUT_CONTROL_DATA[7].st_Title_String := 'Port Security           : <Disable>';

	Xus_TN_INPUT_CONTROL.usa_TN_INPUT_CONTROL_DATA[8].in_Type := INT#02;
	Xus_TN_INPUT_CONTROL.usa_TN_INPUT_CONTROL_DATA[8].in_Y := INT#13;
	Xus_TN_INPUT_CONTROL.usa_TN_INPUT_CONTROL_DATA[8].in_X := INT#44;
	Xus_TN_INPUT_CONTROL.usa_TN_INPUT_CONTROL_DATA[8].by_Attr_mF := BYTE#16#07;
	Xus_TN_INPUT_CONTROL.usa_TN_INPUT_CONTROL_DATA[8].by_Attr_oF := BYTE#16#70;
	Xus_TN_INPUT_CONTROL.usa_TN_INPUT_CONTROL_DATA[8].st_Input_Mask := '       ';
	Xus_TN_INPUT_CONTROL.usa_TN_INPUT_CONTROL_DATA[8].st_Input_Data := 'Disable#Enable';
	Xus_TN_INPUT_CONTROL.usa_TN_INPUT_CONTROL_DATA[8].st_Input_ToolTip := 'Push SPACE to Enable/Disable Access Control for the WEB Interface';
	Xus_TN_INPUT_CONTROL.usa_TN_INPUT_CONTROL_DATA[8].in_Input_Option := INT#02;
	Xus_TN_INPUT_CONTROL.usa_TN_INPUT_CONTROL_DATA[8].in_Title_Y_Offset := INT#00;
	Xus_TN_INPUT_CONTROL.usa_TN_INPUT_CONTROL_DATA[8].in_Title_X_Offset := -27;
	Xus_TN_INPUT_CONTROL.usa_TN_INPUT_CONTROL_DATA[8].by_Title_Attr := BYTE#16#70;
	Xus_TN_INPUT_CONTROL.usa_TN_INPUT_CONTROL_DATA[8].st_Title_String := 'Access Control for Web  : <Disable>';

	Xus_TN_INPUT_CONTROL.usa_TN_INPUT_CONTROL_DATA[9].in_Type := INT#02;
	Xus_TN_INPUT_CONTROL.usa_TN_INPUT_CONTROL_DATA[9].in_Y := INT#14;
	Xus_TN_INPUT_CONTROL.usa_TN_INPUT_CONTROL_DATA[9].in_X := INT#44;
	Xus_TN_INPUT_CONTROL.usa_TN_INPUT_CONTROL_DATA[9].by_Attr_mF := BYTE#16#07;
	Xus_TN_INPUT_CONTROL.usa_TN_INPUT_CONTROL_DATA[9].by_Attr_oF := BYTE#16#70;
	Xus_TN_INPUT_CONTROL.usa_TN_INPUT_CONTROL_DATA[9].st_Input_Mask := '        ';
	Xus_TN_INPUT_CONTROL.usa_TN_INPUT_CONTROL_DATA[9].st_Input_Data := 'Default#Profinet';
	Xus_TN_INPUT_CONTROL.usa_TN_INPUT_CONTROL_DATA[9].st_Input_ToolTip := 'Push SPACE to select the switch operating mode';
	Xus_TN_INPUT_CONTROL.usa_TN_INPUT_CONTROL_DATA[9].in_Input_Option := INT#02;
	Xus_TN_INPUT_CONTROL.usa_TN_INPUT_CONTROL_DATA[9].in_Title_Y_Offset := INT#00;
	Xus_TN_INPUT_CONTROL.usa_TN_INPUT_CONTROL_DATA[9].in_Title_X_Offset := -27;
	Xus_TN_INPUT_CONTROL.usa_TN_INPUT_CONTROL_DATA[9].by_Title_Attr := BYTE#16#70;
	Xus_TN_INPUT_CONTROL.usa_TN_INPUT_CONTROL_DATA[9].st_Title_String := 'Switch Operating Mode   : <Default >';

	Xus_TN_INPUT_CONTROL.usa_TN_INPUT_CONTROL_DATA[10].in_Type := INT#02;
	Xus_TN_INPUT_CONTROL.usa_TN_INPUT_CONTROL_DATA[10].in_Y := INT#16;
	Xus_TN_INPUT_CONTROL.usa_TN_INPUT_CONTROL_DATA[10].in_X := INT#44;
	Xus_TN_INPUT_CONTROL.usa_TN_INPUT_CONTROL_DATA[10].by_Attr_mF := BYTE#16#07;
	Xus_TN_INPUT_CONTROL.usa_TN_INPUT_CONTROL_DATA[10].by_Attr_oF := BYTE#16#70;
	Xus_TN_INPUT_CONTROL.usa_TN_INPUT_CONTROL_DATA[10].st_Input_Mask := '       ';
	Xus_TN_INPUT_CONTROL.usa_TN_INPUT_CONTROL_DATA[10].st_Input_Data := 'Enable#Disable';
	Xus_TN_INPUT_CONTROL.usa_TN_INPUT_CONTROL_DATA[10].st_Input_ToolTip := 'Push SPACE to Enable/Disable Web Interface (effective after reboot)';
	Xus_TN_INPUT_CONTROL.usa_TN_INPUT_CONTROL_DATA[10].in_Input_Option := INT#02;
	Xus_TN_INPUT_CONTROL.usa_TN_INPUT_CONTROL_DATA[10].in_Title_Y_Offset := INT#00;
	Xus_TN_INPUT_CONTROL.usa_TN_INPUT_CONTROL_DATA[10].in_Title_X_Offset := -27;
	Xus_TN_INPUT_CONTROL.usa_TN_INPUT_CONTROL_DATA[10].by_Title_Attr := BYTE#16#70;
	Xus_TN_INPUT_CONTROL.usa_TN_INPUT_CONTROL_DATA[10].st_Title_String := 'Web Interface           : <Enable >';

	Xus_TN_INPUT_CONTROL.usa_TN_INPUT_CONTROL_DATA[11].in_Type := INT#02;
	Xus_TN_INPUT_CONTROL.usa_TN_INPUT_CONTROL_DATA[11].in_Y := INT#17;
	Xus_TN_INPUT_CONTROL.usa_TN_INPUT_CONTROL_DATA[11].in_X := INT#44;
	Xus_TN_INPUT_CONTROL.usa_TN_INPUT_CONTROL_DATA[11].by_Attr_mF := BYTE#16#07;
	Xus_TN_INPUT_CONTROL.usa_TN_INPUT_CONTROL_DATA[11].by_Attr_oF := BYTE#16#70;
	Xus_TN_INPUT_CONTROL.usa_TN_INPUT_CONTROL_DATA[11].st_Input_Mask := '       ';
	Xus_TN_INPUT_CONTROL.usa_TN_INPUT_CONTROL_DATA[11].st_Input_Data := 'Enable#Disable';
	Xus_TN_INPUT_CONTROL.usa_TN_INPUT_CONTROL_DATA[11].st_Input_ToolTip := 'Push SPACE to Enable/Disable Telnet Interface (effective after reboot)';
	Xus_TN_INPUT_CONTROL.usa_TN_INPUT_CONTROL_DATA[11].in_Input_Option := INT#02;
	Xus_TN_INPUT_CONTROL.usa_TN_INPUT_CONTROL_DATA[11].in_Title_Y_Offset := INT#00;
	Xus_TN_INPUT_CONTROL.usa_TN_INPUT_CONTROL_DATA[11].in_Title_X_Offset := -27;
	Xus_TN_INPUT_CONTROL.usa_TN_INPUT_CONTROL_DATA[11].by_Title_Attr := BYTE#16#70;
	Xus_TN_INPUT_CONTROL.usa_TN_INPUT_CONTROL_DATA[11].st_Title_String := 'Telnet Interface        : <Enable >';

	Xus_TN_INPUT_CONTROL.usa_TN_INPUT_CONTROL_DATA[12].in_Type := INT#02;
	Xus_TN_INPUT_CONTROL.usa_TN_INPUT_CONTROL_DATA[12].in_Y := INT#18;
	Xus_TN_INPUT_CONTROL.usa_TN_INPUT_CONTROL_DATA[12].in_X := INT#44;
	Xus_TN_INPUT_CONTROL.usa_TN_INPUT_CONTROL_DATA[12].by_Attr_mF := BYTE#16#07;
	Xus_TN_INPUT_CONTROL.usa_TN_INPUT_CONTROL_DATA[12].by_Attr_oF := BYTE#16#70;
	Xus_TN_INPUT_CONTROL.usa_TN_INPUT_CONTROL_DATA[12].st_Input_Mask := '       ';
	Xus_TN_INPUT_CONTROL.usa_TN_INPUT_CONTROL_DATA[12].st_Input_Data := 'Enable#Disable';
	Xus_TN_INPUT_CONTROL.usa_TN_INPUT_CONTROL_DATA[12].st_Input_ToolTip := 'Push SPACE to Enable/Disable SNMP Interface (effective after reboot)';
	Xus_TN_INPUT_CONTROL.usa_TN_INPUT_CONTROL_DATA[12].in_Input_Option := INT#02;
	Xus_TN_INPUT_CONTROL.usa_TN_INPUT_CONTROL_DATA[12].in_Title_Y_Offset := INT#00;
	Xus_TN_INPUT_CONTROL.usa_TN_INPUT_CONTROL_DATA[12].in_Title_X_Offset := -27;
	Xus_TN_INPUT_CONTROL.usa_TN_INPUT_CONTROL_DATA[12].by_Title_Attr := BYTE#16#70;
	Xus_TN_INPUT_CONTROL.usa_TN_INPUT_CONTROL_DATA[12].st_Title_String := 'SNMP Interface          : <Enable >';

	Xus_TN_INPUT_CONTROL.usa_TN_INPUT_CONTROL_DATA[13].in_Type := INT#02;
	Xus_TN_INPUT_CONTROL.usa_TN_INPUT_CONTROL_DATA[13].in_Y := INT#20;
	Xus_TN_INPUT_CONTROL.usa_TN_INPUT_CONTROL_DATA[13].in_X := INT#44;
	Xus_TN_INPUT_CONTROL.usa_TN_INPUT_CONTROL_DATA[13].by_Attr_mF := BYTE#16#07;
	Xus_TN_INPUT_CONTROL.usa_TN_INPUT_CONTROL_DATA[13].by_Attr_oF := BYTE#16#70;
	Xus_TN_INPUT_CONTROL.usa_TN_INPUT_CONTROL_DATA[13].st_Input_Mask := '                                 ';
	Xus_TN_INPUT_CONTROL.usa_TN_INPUT_CONTROL_DATA[13].st_Input_Data := 'No reset#Reset Switch#Reset Switch to factory defaults';
	Xus_TN_INPUT_CONTROL.usa_TN_INPUT_CONTROL_DATA[13].st_Input_ToolTip := 'Push SPACE to select Reset Option';
	Xus_TN_INPUT_CONTROL.usa_TN_INPUT_CONTROL_DATA[13].in_Input_Option := INT#02;
	Xus_TN_INPUT_CONTROL.usa_TN_INPUT_CONTROL_DATA[13].in_Title_Y_Offset := INT#00;
	Xus_TN_INPUT_CONTROL.usa_TN_INPUT_CONTROL_DATA[13].in_Title_X_Offset := -27;
	Xus_TN_INPUT_CONTROL.usa_TN_INPUT_CONTROL_DATA[13].by_Title_Attr := BYTE#16#70;
	Xus_TN_INPUT_CONTROL.usa_TN_INPUT_CONTROL_DATA[13].st_Title_String := 'Reset                   : <No reset                         >';

	Xus_TN_INPUT_CONTROL.usa_TN_INPUT_CONTROL_DATA[14].in_Type := INT#02;
	Xus_TN_INPUT_CONTROL.usa_TN_INPUT_CONTROL_DATA[14].in_Y := INT#22;
	Xus_TN_INPUT_CONTROL.usa_TN_INPUT_CONTROL_DATA[14].in_X := INT#18;
	Xus_TN_INPUT_CONTROL.usa_TN_INPUT_CONTROL_DATA[14].by_Attr_mF := BYTE#16#07;
	Xus_TN_INPUT_CONTROL.usa_TN_INPUT_CONTROL_DATA[14].by_Attr_oF := BYTE#16#70;
	Xus_TN_INPUT_CONTROL.usa_TN_INPUT_CONTROL_DATA[14].st_Input_ToolTip := 'Apply and save ALL changes to permanent memory';
	Xus_TN_INPUT_CONTROL.usa_TN_INPUT_CONTROL_DATA[14].in_Input_Option := INT#01;
	Xus_TN_INPUT_CONTROL.usa_TN_INPUT_CONTROL_DATA[14].in_Title_Y_Offset := INT#00;
	Xus_TN_INPUT_CONTROL.usa_TN_INPUT_CONTROL_DATA[14].in_Title_X_Offset := INT#00;
	Xus_TN_INPUT_CONTROL.usa_TN_INPUT_CONTROL_DATA[14].by_Title_Attr := BYTE#16#70;
	Xus_TN_INPUT_CONTROL.usa_TN_INPUT_CONTROL_DATA[14].st_Title_String := '';
	Xus_TN_INPUT_CONTROL.usa_TN_INPUT_CONTROL_DATA[14].st_Input_Mask := '    ';
	Xus_TN_INPUT_CONTROL.usa_TN_INPUT_CONTROL_DATA[14].st_Input_Data := 'SAVE';

	Xus_TN_INPUT_CONTROL.usa_TN_INPUT_CONTROL_DATA[15].in_Type := INT#02;
	Xus_TN_INPUT_CONTROL.usa_TN_INPUT_CONTROL_DATA[15].in_Y := INT#22;
	Xus_TN_INPUT_CONTROL.usa_TN_INPUT_CONTROL_DATA[15].in_X := INT#11;
	Xus_TN_INPUT_CONTROL.usa_TN_INPUT_CONTROL_DATA[15].by_Attr_mF := BYTE#16#07;
	Xus_TN_INPUT_CONTROL.usa_TN_INPUT_CONTROL_DATA[15].by_Attr_oF := BYTE#16#70;
	Xus_TN_INPUT_CONTROL.usa_TN_INPUT_CONTROL_DATA[15].st_Input_ToolTip := 'Apply changes';
	Xus_TN_INPUT_CONTROL.usa_TN_INPUT_CONTROL_DATA[15].in_Input_Option := INT#01;
	Xus_TN_INPUT_CONTROL.usa_TN_INPUT_CONTROL_DATA[15].in_Title_Y_Offset := INT#00;
	Xus_TN_INPUT_CONTROL.usa_TN_INPUT_CONTROL_DATA[15].in_Title_X_Offset := INT#00;
	Xus_TN_INPUT_CONTROL.usa_TN_INPUT_CONTROL_DATA[15].by_Title_Attr := BYTE#16#70;
	Xus_TN_INPUT_CONTROL.usa_TN_INPUT_CONTROL_DATA[15].st_Title_String := '';
	Xus_TN_INPUT_CONTROL.usa_TN_INPUT_CONTROL_DATA[15].st_Input_Mask := '     ';
	Xus_TN_INPUT_CONTROL.usa_TN_INPUT_CONTROL_DATA[15].st_Input_Data := 'APPLY';

	Xus_TN_INPUT_CONTROL.usa_TN_INPUT_CONTROL_DATA[16].in_Type := INT#02;
	Xus_TN_INPUT_CONTROL.usa_TN_INPUT_CONTROL_DATA[16].in_Y := INT#22;
	Xus_TN_INPUT_CONTROL.usa_TN_INPUT_CONTROL_DATA[16].in_X := INT#03;
	Xus_TN_INPUT_CONTROL.usa_TN_INPUT_CONTROL_DATA[16].by_Attr_mF := BYTE#16#07;
	Xus_TN_INPUT_CONTROL.usa_TN_INPUT_CONTROL_DATA[16].by_Attr_oF := BYTE#16#70;
	Xus_TN_INPUT_CONTROL.usa_TN_INPUT_CONTROL_DATA[16].st_Input_ToolTip := 'Return to Main Menu';
	Xus_TN_INPUT_CONTROL.usa_TN_INPUT_CONTROL_DATA[16].in_Input_Option := INT#01;
	Xus_TN_INPUT_CONTROL.usa_TN_INPUT_CONTROL_DATA[16].in_Title_Y_Offset := INT#00;
	Xus_TN_INPUT_CONTROL.usa_TN_INPUT_CONTROL_DATA[16].in_Title_X_Offset := INT#00;
	Xus_TN_INPUT_CONTROL.usa_TN_INPUT_CONTROL_DATA[16].by_Title_Attr := BYTE#16#70;
	Xus_TN_INPUT_CONTROL.usa_TN_INPUT_CONTROL_DATA[16].st_Title_String := '';
	Xus_TN_INPUT_CONTROL.usa_TN_INPUT_CONTROL_DATA[16].st_Input_Mask := '      ';
	Xus_TN_INPUT_CONTROL.usa_TN_INPUT_CONTROL_DATA[16].st_Input_Data := 'LOGOUT';

	(* Control-Tool-Tip *)
	Xus_TN_INPUT_CONTROL.in_ToolTip_Y := INT#23;
	Xus_TN_INPUT_CONTROL.in_ToolTip_X := INT#00;
	Xus_TN_INPUT_CONTROL.by_ToolTip_Attr := BYTE#07;
	Xus_TN_INPUT_CONTROL.in_ToolTip_Size := INT#80;

	(* Control-Verwaltung initialisieren *)
	Xus_TN_INPUT_CONTROL.in_Count := INT#16;
	Xus_TN_INPUT_CONTROL.bo_Enable := TRUE;
	Xus_TN_INPUT_CONTROL.bo_Reset_Fokus := TRUE;

END_IF;

IF (Xus_TN_SCREEN.in_Page_Number = INT#05) THEN

	(* eingegebenen String übernehmen *)
	IF Xus_TN_INPUT_CONTROL.usa_TN_INPUT_CONTROL_DATA[16].bo_Input_Entered = TRUE THEN

		Xus_TN_INPUT_CONTROL.usa_TN_INPUT_CONTROL_DATA[16].bo_Input_Entered := FALSE;
		Xus_TN_SCREEN.in_Page_Number := INT#00;
	END_IF;
END_IF;
END_PROGRAM

(* POU WORLD_WEATHER_DEMO, CFC *)
PROGRAM WORLD_WEATHER_DEMO
VAR
	IP_C: IP_C;
	S_BUF: NETWORK_BUFFER;
	R_BUF: NETWORK_BUFFER;
	IP_CONTROL_1: IP_CONTROL;
	activate: BOOL := TRUE;
	done: BOOL;
	busy: BOOL;
	error_c: DWORD;
	error_t: BYTE;
	latitude: REAL := 48.21;
	longitude: REAL := 16.37;
	WORLD_WEATHER: WORLD_WEATHER;
	WW_DATA: WORLD_WEATHER_DATA;
	CLK_PRG: CLK_PRG;
	WORLD_WEATHER_DESC_GE: WORLD_WEATHER_DESC_GE;
	WORLD_WEATHER_ICON_OSCAT: WORLD_WEATHER_ICON_OSCAT;
END_VAR
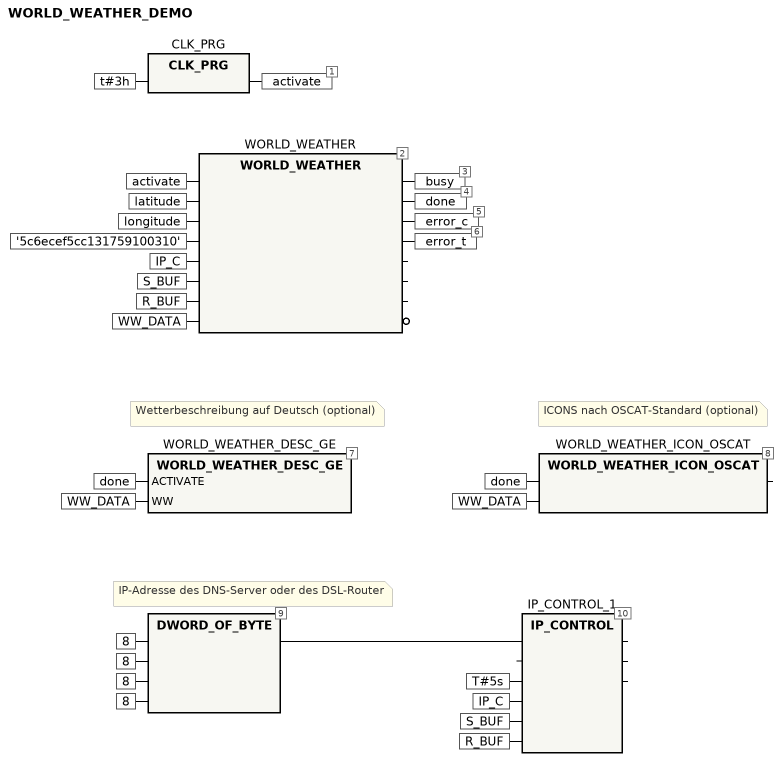
_CFC_ (* Continuous Function Chart, elements in execution order *)
#0 CLK_PRG:CLK_PRG(t#3h)
#1 activate <= #0
#2 WORLD_WEATHER:WORLD_WEATHER(activate, latitude, longitude, '5c6ecef5cc131759100310', IP_C, S_BUF, R_BUF, WW_DATA)
#3 busy <= #2.out 1
#4 done <= #2.out 2
#5 error_c <= #2.out 3
#6 error_t <= #2.out 4
#7 WORLD_WEATHER_DESC_GE:WORLD_WEATHER_DESC_GE(ACTIVATE: done, WW: WW_DATA)
#8 WORLD_WEATHER_ICON_OSCAT:WORLD_WEATHER_ICON_OSCAT(done, WW_DATA)
#9 DWORD_OF_BYTE(8, 8, 8, 8)
#10 IP_CONTROL_1:IP_CONTROL(#9, -, T#5s, IP_C, S_BUF, R_BUF)
(* ICONS nach OSCAT-Standard (optional) *)
(* IP-Adresse des DNS-Server oder des DSL-Router *)
(* Wetterbeschreibung auf Deutsch (optional) *)
_END_CFC_
END_PROGRAM

(* POU WORLD_WEATHER, ST *)
FUNCTION_BLOCK WORLD_WEATHER
VAR_IN_OUT
	IP_C : IP_C; (* IP_Control Verwaltungsstruktur *)
	S_BUF : NETWORK_BUFFER;
	R_BUF : NETWORK_BUFFER;
	WW : WORLD_WEATHER_DATA;
END_VAR
VAR_INPUT
	ACTIVATE : BOOL;
	LATITUDE : REAL;
	LONGITUDE : REAL;
	KEY : STRING(30);
END_VAR
VAR_OUTPUT
	BUSY : BOOL;
	DONE : BOOL;
	ERROR_C : DWORD;
	ERROR_T : BYTE;
END_VAR
VAR
	URL_DATA : url;
	DNS_CLIENT : DNS_CLIENT;
	HTTP_GET : HTTP_GET;
	CPB : CSV_PARSER_BUF;
	last_state : BOOL;
	value_int : INT;
	value_real : REAL;
	v_real : REAL;
	state : INT;
	url_str : STRING(STRING_LENGTH);
	offset : UDINT;
	size : INT;
	sep : BYTE;
	cnt : INT;
	day : INT;
	idx : INT;
	run : BYTE;
	result : BYTE;
	value : STRING(STRING_LENGTH);
	pos : INT;
END_VAR

(*

version 1.4	05. oct 2012
programmer 	ks
tested by	ks

WORLD_WEATHER lädt von worldweather.com eine Wetter csv-datei und analysiert die Daten und legt diese in einem Array ab
Die Wetterdaten werden für 5 tage aufbereitet

*)
CASE state OF

00:
	IF ACTIVATE AND NOT last_state THEN
		state := 20;
		DONE := FALSE;
		BUSY := TRUE;
		ERROR_C := DWORD#0;
		ERROR_T := BYTE#0;
	END_IF;

20: (* URL for DNS UND HTTP-GET *)
	(* Example: http://free.worldweatheronline.com/feed/weather.ashx?q=48.21,16.37&format=csv&num_of_days=5&key=xxxxxxxxxxxxxxxxxxxxxx *)
	url_str := CONCAT('http://free.worldweatheronline.com/feed/weather.ashx?q=',REAL_TO_STRF(LATITUDE,6,D:='.'));
	url_str := CONCAT(url_str,',');
	url_str := CONCAT(url_str,REAL_TO_STRF(LONGITUDE,6,D:='.'));
	url_str := CONCAT(url_str,'&format=csv&num_of_days=5&key=');
	url_str := CONCAT(url_str,key);

	URL_DATA:=STRING_TO_URL(STR:=url_str, DEFAULT_PROTOCOL:='', DEFAULT_PATH:='' );
	state := 40;

40:
	IF DNS_CLIENT.DONE THEN
		state := 60;
	ELSIF (DNS_CLIENT.ERROR > DWORD#00) THEN
		(* Fehlerbehandlung *)
		ERROR_C := DNS_CLIENT.ERROR;
	ERROR_T := BYTE#01;
		state   := 100;
	END_IF;

60:
	IF HTTP_GET.DONE THEN
		sep := 0;
		idx := 0;
		day := 0;
		cnt := 0;
		OFFSET := HTTP_GET.BODY_START; (* Start Offset vorgeben *)
		size := HTTP_GET.BODY_STOP; (* End Position *)
		run := 1; (* Element suchen *)
		state := 80;

	ELSIF (HTTP_GET.ERROR > DWORD#00) THEN
		(* Fehlerbehandlung *)
		ERROR_C := HTTP_GET.ERROR;
		ERROR_T := BYTE#02;
		state := 100;
	END_IF;

80:	IF run = 0 THEN (* kein Befehl mehr aktiv ? *)
		run := 1; (*  nächstes Element suchen  *)
		IF result = 1 OR result = 2 THEN
			value_int := 0;
			value_real := 0.0;
			(* automatische konvertierung in real und int ausführen *)
			IF LEN(value) <= 20 THEN
				v_real:=FLOAT_TO_REAL(FLT:=value);
				IF CHK_REAL(v_real) = 0 THEN (* !!! prüft auf gültigen REAL Wert, ansonsten stürzt Twincat ab !!!!  *)
					value_real := v_real;
					value_int := REAL_TO_INT(value_real);
				END_IF;
			END_IF;
			cnt := cnt + 1;


			IF cnt = 1 AND LEFT(value,1) <> '#' THEN
				cnt := 0;
			END_IF;

			IF cnt >=8 AND cnt <= 87 THEN
				IF cnt > 22 THEN
					CASE idx OF
					00:	WW.DAY[day].DATE_OF_DAY := value;
					01:	WW.DAY[day].TEMP_MAX_C := value_int;
					02:	WW.DAY[day].TEMP_MAX_F := value_int;
					03:	WW.DAY[day].TEMP_MIN_C := value_int;
					04:	WW.DAY[day].TEMP_MIN_F := value_int;
					05:	WW.DAY[day].WIND_SPEED_MILES := value_int;
					06:	WW.DAY[day].WIND_SPEED_KMPH := value_int;
					07:	WW.DAY[day].WIND_DIR_DEGREE := value_int;
					08:	WW.DAY[day].WIND_DIR16POINT := value;
					09:	WW.DAY[day].WEATHER_CODE := value_int;
					10:	pos := FIND(value, '/wsymbol_');
						WW.DAY[day].WEATHER_ICON := DEC_TO_INT(MID(value,4,pos+9));
					11:	WW.DAY[day].WEATHER_DESC := value;
					12:	WW.DAY[day].PRECIPMM := value_real;
					END_CASE;
					idx := idx + 1;
					IF idx > 12 THEN
						idx := 0;
						day := day + 1;
					END_IF;
				ELSE
					CASE cnt OF
					08:	sep :=44; (* ab jetzt mit Trennzeichen arbeiten, *)
					09:	WW.CUR.OBSERVATION_TIME := value;
					10:	WW.CUR.TEMP_C := value_int;
					11:	WW.CUR.WEATHER_CODE := value_int;
					12:	pos := FIND(value, '/wsymbol_');
						WW.CUR.WEATHER_ICON := DEC_TO_INT(MID(value,4,pos+9));
					13:	WW.CUR.WEATHER_DESC := value;
					14:	WW.CUR.WIND_SPEED_MILES := value_int;
					15:	WW.CUR.WIND_SPEED_KMPH := value_int;
					16:	WW.CUR.WIND_DIR_DEGREE := value_int;
					17:	WW.CUR.WIND_DIR16POINT := value;
					18:	WW.CUR.PRECIPMM := value_real;
					19:	WW.CUR.HUMIDITY := value_int;
					20:	WW.CUR.VISIBILITY := value_int;
					21:	WW.CUR.PRESSURE := value_int;
					22:	WW.CUR.CLOUDOVER := value_int;
					END_CASE;
				END_IF;
			END_IF;
		ELSIF result = 10 THEN (* nichts mehr gefunden *)
			DONE  := TRUE;
			run := 0; (* Auswertung beenden *)
			state := 100;
		END_IF;
	END_IF;

100:
	(* UNLOCK HTTP DATA *)
	IF (NOT HTTP_GET.DONE) THEN
		state := 0;
		BUSY := FALSE;
		DONE := ERROR_T = BYTE#0;
	END_IF;

END_CASE;

(* ---------------- DNS --------------- *)
DNS_CLIENT(	IP_C:=IP_C,
			S_BUF:=S_BUF,
			R_BUF:=R_BUF,
			DOMAIN:=URL_DATA.DOMAIN,
			IP4_DNS:=DWORD#00,
			ACTIVATE:=state=40 (* DNS Start *)
			);
(* nicht oder nicht direkt verwendete Parameter *)
(*	DWORD :=DNS_CLIENT.IP4;
	BOOL  :=DNS_CLIENT.DONE;
	BYTE  :=DNS_CLIENT.ERROR; *)
(* -------------------------------------*)

(* ------------- HTTP_GET --------------- *)
HTTP_GET(	IP_C:=IP_C,
			S_BUF:=S_BUF,
			R_BUF:=R_BUF,
			IP4:=DNS_CLIENT.IP4,
			GET:=state=60,
			MODE:=BYTE#2, (* HTTP 1.1 mit persistenter Verbindung *)
			UNLOCK_BUF:=state=100,
			URL_DATA:=URL_DATA
			);

(* nicht oder nicht direkt verwendete Parameter *)
(*	STRING := HTTP_GET.HTTP_STATUS;
	UINT :=HTTP_GET.HEADER_START;
	UINT :=HTTP_GET.HEADER_STOP;
	UINT :=HTTP_GET.BODY_START;
	UINT :=HTTP_GET.BODY_STOP;
	BOOL :=HTTP_GET.DONE;
	BYTE :=HTTP_GET.ERROR;
*)
(* -------------------------------------*)
CPB(SEP:=sep,RUN:=run,OFFSET:=OFFSET,VALUE:=value,PT:=R_BUF,RESULT=>result); (* CSV PARAMETER BUF *)

last_state := ACTIVATE;

(* revision history
ks	01.oct. 2010	rev 1.0
	original version

ks	01.feb. 2011	rev 1.1
	rücksetzen von cnt 

ks	07.apr. 2011	rev 1.2
	neue Domain "free.worldweatheronline.com" (Ab 30.04.2011 notwendig)

ks	05.jan. 2012	rev 1.3
	neues datenelement "icon" integriert, REAL_TO_STRF parameter D

ks	05.oct. 2012	rev 1.4
	workaround für chunked html data

*)
END_FUNCTION_BLOCK

(* POU WORLD_WEATHER_DESC_GE, ST *)
FUNCTION_BLOCK WORLD_WEATHER_DESC_GE
VAR_IN_OUT
	WW : WORLD_WEATHER_DATA;
END_VAR
VAR_INPUT
	ACTIVATE : BOOL;
END_VAR
VAR
	act_last : BOOL;
	x : INT;
	y : INT;
	str : STRING(60);
	i : INT;
END_VAR

(*

version 1.0		04. may. 2011
programmer 		ks
tested by			ks

WORLD_WEATHER_DESC_GE ändert die englischen Wetterbeschreibungstexte auf deutsche Texte um
*)
IF ACTIVATE AND act_last = FALSE THEN
	i := 0;
	FOR y := 1 TO 12 DO
		CASE y OF
		1,3,5,7,9:		x :=  WW.DAY[i].WEATHER_CODE;
		2,4,6,8,10:	WW.DAY[i].WEATHER_DESC := str;
					i := i + 1;
		11:			x :=  WW.CUR.WEATHER_CODE;
		12:			WW.CUR.WEATHER_DESC := str;
		END_CASE;

		CASE x OF
			113	:	str := 'heiter/sonnig';
			116	:	str := 'stellenweise wolkig';
			119	:	str := 'wolkig';
			122	:	str := 'bewölkt';
			143	:	str := 'Nebel';
			176	:	str := 'stellenweise nahegelegener Regen';
			179	:	str := 'stellenweise nahegelegener Schneefall';
			182	:	str := 'stellenweise nahegelegener Eisregen';
			185	:	str := 'stellenweise gefrierender Niesel';
			200	:	str := 'nahegelegene Sturm';
			227	:	str := 'Schneetreiben';
			230	:	str := 'Schneesturm';
			248	:	str := 'Nebel';
			260	:	str := 'gefrierender Nebel';
			263	:	str := 'stellenweise leichter Nieselregen';
			266	:	str := 'leichter Niesel';
			281	:	str := 'gefrierender Nieselregen';
			284	:	str := 'stark gefrierender Nieselregen';
			293	:	str := 'stellenweise leichter Regen';
			296	:	str := 'leichter Regen';
			299	:	str := 'zeitweise etwas Regen';
			302	:	str := 'mäßiger Regen';
			305	:	str := 'zeitweise etwas starker Regen';
			308	:	str := 'starker Regen';
			311	:	str := 'leichter gefrierender Regen';
			314	:	str := 'mäßiger oder starker Eisregen';
			317	:	str := 'leichter Eisregen';
			320	:	str := 'mäßiger oder starker Eisregen';
			323	:	str := 'stellenweise leichter Schneefall';
			326	:	str := 'leichter Scheefall';
			329	:	str := 'stellenweise moderater Schneefall';
			332	:	str := 'mäßiger Schnee';
			335	:	str := 'stellenweise starker Scheefall';
			338	:	str := 'starker Schneefall';
			350	:	str := 'Hagel';
			353	:	str := 'leichte Regenfälle';
			356	:	str := 'mäßiger oder starker Regenfall';
			359	:	str := 'sintflutartige Regenfälle';
			362	:	str := 'leichter Eisregen';
			365	:	str := 'mäßiger oder starker Eisregen';
			368	:	str := 'leichte Schneeschauer';
			371	:	str := 'mäßiger oder starker Schneefall';
			374	:	str := 'leichter Hagel';
			377	:	str := 'mäßiger oder starker Hagel';
			386	:	str := 'stellenweise leichter Regen in Gewittergebiet';
			389	:	str := 'mäßiger oder starker Regen in Gewittergebiet';
			392	:	str := 'stellenweise leichter Schneefall in Gewittergebiet';
			395	:	str := 'mäßiger oder starker Schnee in Gewittergebiet';
		ELSE
			str := 	'nicht verfügbar';
		END_CASE;
	END_FOR;
END_IF;
act_last := ACTIVATE;

(* revision history
ks	04. may. 2011	rev 1.0
	original version
*)
END_FUNCTION_BLOCK

(* POU WORLD_WEATHER_ICON_OSCAT, ST *)
FUNCTION_BLOCK WORLD_WEATHER_ICON_OSCAT
VAR_IN_OUT
	WW : WORLD_WEATHER_DATA;
END_VAR
VAR_INPUT
	ACTIVATE : BOOL;
END_VAR
VAR
	dat : ARRAY[0..41] OF INT := 0,14,12,9,9,0,7,7,0,2,2,3,3,1,0,0,17,4,4,3,3,1,0,0,17,2,2,3,3,1,0,0,17,2,4,3,3,1,0,0,17,0;
	act_last : BOOL;
	x : INT;
	i : INT;
END_VAR

(*

version 1.0		04. may. 2011
programmer 		ks
tested by			ks

WORLD_WEATHER_ICON_OSCAT ändert die ICON Nummer auf den OSCAT-Standard um
*)
IF ACTIVATE AND act_last = FALSE THEN
	x := LIMIT(0,WW.CUR.WEATHER_ICON,41);
	WW.CUR.WEATHER_ICON := dat[x];
	FOR i := 0 TO 4 DO
		x := LIMIT(0,WW.DAY[i].WEATHER_ICON,41);
		WW.DAY[i].WEATHER_ICON := dat[x];
	END_FOR;
END_IF;
act_last := ACTIVATE;

(* revision history
ks	04. may. 2011	rev 1.0
	original version
*)
END_FUNCTION_BLOCK

(* POU YAHOO_WEATHER_DEMO, CFC *)
PROGRAM YAHOO_WEATHER_DEMO
VAR
	IP_C: IP_C;
	S_BUF: NETWORK_BUFFER;
	R_BUF: NETWORK_BUFFER;
	IP_CONTROL_1: IP_CONTROL;
	activate: BOOL;
	done: BOOL;
	busy: BOOL;
	error_c: DWORD;
	error_t: BYTE;
	YAHOO_WEATHER: YAHOO_WEATHER;
	YW_DATA: YAHOO_WEATHER_DATA;
	CLK_PRG: CLK_PRG;
	YAHOO_WEATHER_DESC_GE: YAHOO_WEATHER_DESC_GE;
	YAHOO_WEATHER_ICON_OSCAT: YAHOO_WEATHER_ICON_OSCAT;
END_VAR
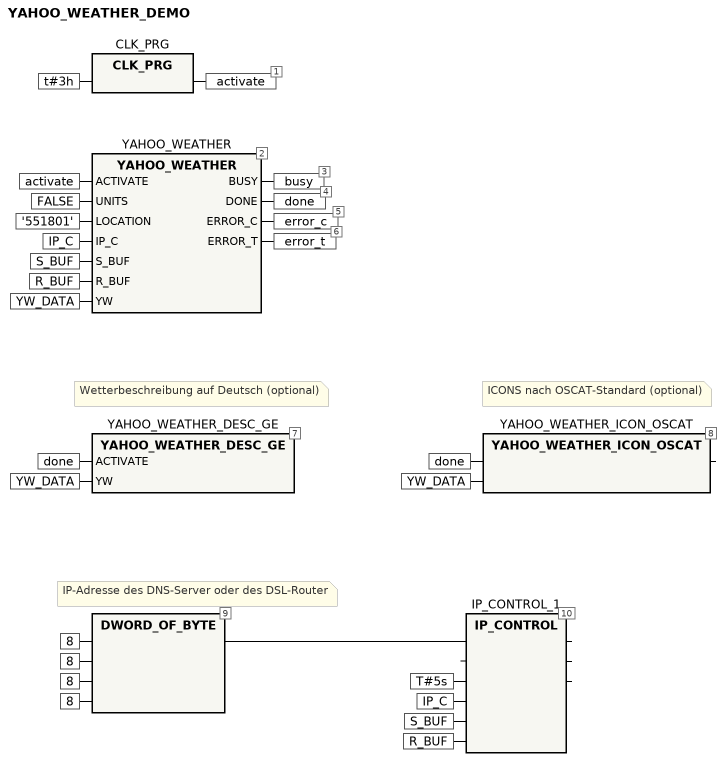
_CFC_ (* Continuous Function Chart, elements in execution order *)
#0 CLK_PRG:CLK_PRG(t#3h)
#1 activate <= #0
#2 YAHOO_WEATHER:YAHOO_WEATHER(ACTIVATE: activate, UNITS: FALSE, LOCATION: '551801', IP_C: IP_C, S_BUF: S_BUF, R_BUF: R_BUF, YW: YW_DATA)
#3 busy <= #2.BUSY
#4 done <= #2.DONE
#5 error_c <= #2.ERROR_C
#6 error_t <= #2.ERROR_T
#7 YAHOO_WEATHER_DESC_GE:YAHOO_WEATHER_DESC_GE(ACTIVATE: done, YW: YW_DATA)
#8 YAHOO_WEATHER_ICON_OSCAT:YAHOO_WEATHER_ICON_OSCAT(done, YW_DATA)
#9 DWORD_OF_BYTE(8, 8, 8, 8)
#10 IP_CONTROL_1:IP_CONTROL(#9, -, T#5s, IP_C, S_BUF, R_BUF)
(* ICONS nach OSCAT-Standard (optional) *)
(* IP-Adresse des DNS-Server oder des DSL-Router *)
(* Wetterbeschreibung auf Deutsch (optional) *)
_END_CFC_
END_PROGRAM

(* POU YAHOO_WEATHER, ST *)
FUNCTION_BLOCK YAHOO_WEATHER
VAR_IN_OUT
	IP_C : IP_C; (* IP_Control Verwaltungsstruktur *)
	S_BUF : NETWORK_BUFFER;
	R_BUF : NETWORK_BUFFER;
	YW : YAHOO_WEATHER_DATA;
END_VAR
VAR_INPUT
	ACTIVATE : BOOL;
	UNITS : BOOL;
	LOCATION : STRING(20);
END_VAR
VAR_OUTPUT
	BUSY : BOOL;
	DONE : BOOL;
	ERROR_C : DWORD;
	ERROR_T : BYTE;
END_VAR
VAR
	CTRL : XML_CONTROL;
	XML_READER : XML_READER;
	URL_DATA : url;
	DNS_CLIENT : DNS_CLIENT;
	HTTP_GET : HTTP_GET;
	last_state : BOOL;
	value_int : INT;
	value_real : REAL;
	v_real : REAL;
	state : INT;
END_VAR

(*

version 1.3		04. may. 2011
programmer 		ks
tested by			ks

YAHOO_WEATHER lädt vom Yahoo-Webserver einen Wetter RSS-Feed und analysiert die Daten und legt diese in einem Array ab
*)
CASE state OF

00:	IF ACTIVATE AND NOT last_state THEN
		state := 20;
		DONE := FALSE;
		BUSY := TRUE;
		ERROR_C := DWORD#0;
		ERROR_T := BYTE#0;
	END_IF;

20: (* URL for DNS UND HTTP-GET *)
	(* Example: http://weather.yahooapis.com/forecastrss?p=94089&u=c *)
	URL_DATA:=STRING_TO_URL(STR:='http://weather.yahooapis.com/forecastrss',
							DEFAULT_PROTOCOL:='',
							DEFAULT_PATH:=''
							);
  	URL_DATA.QUERY := CONCAT('w=',LOCATION);

	IF UNITS THEN
		URL_DATA.QUERY := CONCAT(URL_DATA.QUERY,'&u=f'); (* fahrenheit *)
	ELSE
		URL_DATA.QUERY := CONCAT(URL_DATA.QUERY,'&u=c'); (* celsius *)
	END_IF;
	state := 40;

40:	IF DNS_CLIENT.DONE THEN
		state := 60;
	ELSIF (DNS_CLIENT.ERROR > DWORD#00) THEN
		(* Fehlerbehandlung *)
		ERROR_C := DNS_CLIENT.ERROR;
	ERROR_T := BYTE#01;
		state   := 100;
	END_IF;

60:	IF HTTP_GET.DONE THEN
		state := 80;
		CTRL.START_POS := HTTP_GET.BODY_START;
		CTRL.STOP_POS := HTTP_GET.BODY_STOP;
		CTRL.COMMAND := WORD#2#10000000_00011000; (* ONLY TEXT AND ATTRIBUTE *)
		CTRL.WATCHDOG  := T#1ms;

	ELSIF (HTTP_GET.ERROR > DWORD#00) THEN
		(* Fehlerbehandlung *)
		ERROR_C := HTTP_GET.ERROR;
		ERROR_T := BYTE#02;
		state := 100;
	END_IF;

80: XML_READER(CTRL:=CTRL,BUF:=R_BUF.BUFFER); (* XML Daten seriell lesen *)
	IF CTRL.TYP < 98 THEN (* nur auswerten wenn kein Watchdog durchlauf *)
		value_int := 0;
		value_real := 0.0;
		(* automatische konvertierung in real und int ausführen *)
		IF LEN(CTRL.VALUE) <= 20 THEN
			v_real:=FLOAT_TO_REAL(FLT:=CTRL.VALUE);
			IF CHK_REAL(v_real) = 0 THEN (* !!! prüft auf gültigen REAL Wert, ansonsten stürzt Twincat ab !!!!  *)
				value_real := v_real;
				value_int := REAL_TO_INT(value_real);
			END_IF;
		END_IF;

		IF CTRL.COUNT < UINT#52 THEN (* Performance-Teilung *)
			(* ------------ Teil 1 --------------*)
			CASE UINT_TO_INT(CTRL.COUNT) OF
			027: YW.TimeToLive := value_int;
			030: YW.location_city := CTRL.VALUE;
			031: YW.location_region := CTRL.VALUE;
			032: YW.location_country := CTRL.VALUE;
			035: YW.unit_temperature := CTRL.VALUE;
			036: YW.unit_distance := CTRL.VALUE;
			037: YW.unit_pressure := CTRL.VALUE;
			038: YW.unit_speed := CTRL.VALUE;
			041: YW.wind_chill := value_int;
			042: YW.wind_direction := value_int;
			043: YW.wind_speed := value_real;
			046: YW.atmosphere_humidity := value_int;
			047: YW.atmosphere_visibility := value_real;
			048: YW.atmosphere_pressure := value_int;
			049: YW.atmosphere_rising := value_int;
			END_CASE;
		ELSE
			(* ------------ Teil 2 --------------*)
			CASE UINT_TO_INT(CTRL.COUNT) OF
			052: YW.astronomy_sunrise := CTRL.VALUE;
			053: YW.astronomy_sunset := CTRL.VALUE;
			077: YW.geo_latitude := value_real;
			080: YW.geo_longitude := value_real;
			089: YW.cur_conditions_text := CTRL.VALUE;
			090: YW.cur_conditions_code := value_int;
				YW.cur_conditions_icon := value_int;
			091: YW.cur_conditions_temp := value_int;
			100: YW.forcast_today_low_temp := value_int;
			101: YW.forcast_today_high_temp := value_int;
			102: YW.forcast_today_text := CTRL.VALUE;
			103: YW.forcast_today_code := value_int;
				YW.forcast_today_icon := value_int;
			108: YW.forcast_tomorrow_low_temp := value_int;
			109: YW.forcast_tomorrow_high_temp := value_int;
			110: YW.forcast_tomorrow_text := CTRL.VALUE;
			111: YW.forcast_tomorrow_code := value_int;
				YW.forcast_tomorrow_icon := value_int;
			END_CASE;
		END_IF;
	ELSIF CTRL.TYP = 99 THEN (* EXIT - letztes Element gelesen *)
		DONE  := TRUE;
		state := 100;
	END_IF; 

100:
	(* UNLOCK HTTP DATA *)
	IF (NOT HTTP_GET.DONE) THEN
		state := 0;
		BUSY := FALSE;
		DONE := ERROR_T = BYTE#0;
	END_IF; 

	END_CASE;

(* ---------------- DNS --------------- *)
DNS_CLIENT(	IP_C:=IP_C,
			S_BUF:=S_BUF,
			R_BUF:=R_BUF,
			DOMAIN:=URL_DATA.DOMAIN,
			IP4_DNS:=DWORD#00,
			ACTIVATE:=state=40 (* DNS Start *)
			);
(* nicht oder nicht direkt verwendete Parameter *)
(*	DWORD :=DNS_CLIENT.IP4;
	BOOL  :=DNS_CLIENT.DONE;
	BYTE  :=DNS_CLIENT.ERROR; *)
(* -------------------------------------*)

(* ------------- HTTP_GET --------------- *)
HTTP_GET(	IP_C:=IP_C,
			S_BUF:=S_BUF,
			R_BUF:=R_BUF,
			IP4:=DNS_CLIENT.IP4,
			GET:=state=60,
			MODE:=BYTE#2, (* HTTP 1.1 mit persistenter Verbindung *)
			UNLOCK_BUF:=state=100,
			URL_DATA:=URL_DATA
			);

(* nicht oder nicht direkt verwendete Parameter *)
(*	STRING := HTTP_GET.HTTP_STATUS;
	UINT :=HTTP_GET.HEADER_START;
	UINT :=HTTP_GET.HEADER_STOP;
	UINT :=HTTP_GET.BODY_START;
	UINT :=HTTP_GET.BODY_STOP;
	BOOL :=HTTP_GET.DONE;
	BYTE :=HTTP_GET.ERROR;
*)
(* -------------------------------------*)

last_state := ACTIVATE;

(* revision history
ks	18. dez. 2008	rev 1.0
	original version

ks	01. oct. 2009	rev 1.1
	YAHOO_WEATHER_DATA

ks	24. sep. 2010	rev 1.2
	new URL-Location-parameter and REAL_CHECK (TwinCat BUG) 

ks	04. may. 2011	rev 1.3
	neue elemente:  CUR_CONDITIONS_ICON, FORCAST_TODAY_ICON, FORCAST_TOMORROW_ICON

*)
END_FUNCTION_BLOCK

(* POU YAHOO_WEATHER_DESC_GE, ST *)
FUNCTION_BLOCK YAHOO_WEATHER_DESC_GE
VAR_IN_OUT
	YW : YAHOO_WEATHER_DATA;
END_VAR
VAR_INPUT
	ACTIVATE : BOOL;
END_VAR
VAR
	act_last : BOOL;
	x : INT;
	y : INT;
	str : STRING(40);
END_VAR

(*

version 1.0		04. may. 2011
programmer 		ks
tested by			ks

YAHOO_WEATHER_DESC_GE ändert die englischen Wetterbeschreibungstexte auf deutsche Texte um
*)
IF ACTIVATE AND act_last = FALSE THEN
	FOR y := 1 TO 4 DO
		CASE y OF
		1:	x := YW.CUR_CONDITIONS_CODE;
		2 :	YW.CUR_CONDITIONS_TEXT := str;
			x := YW.FORCAST_TODAY_CODE;
		3 :	YW.FORCAST_TODAY_TEXT := str;
			x := YW.FORCAST_TOMORROW_CODE;
		4 :	YW.FORCAST_TOMORROW_TEXT := str;
		END_CASE;

		CASE x OF
		00:	str := 'Wirbelsturm';
		01:	str := 'Tropensturm';
		02:	str := 'Wirbelsturm';
		03:	str := 'starkes Gewitter ';
		04:	str := 'Gewitter';
		05:	str := 'Schneeregen';
		06:	str := 'Schneeregen';
		07:	str := 'Schneeregen';
		08:	str := 'gefrierender Nieselregen';
		09:	str := 'Nieselregen';
		10:	str := 'gefrierender Regen';
		11:	str := 'Regenfälle';
		12:	str := 'Regenfälle';
		13:	str := 'Schneegestöber';
		14:	str := 'leichte Schneefälle';
		15:	str := 'Schneetreiben';
		16:	str := 'Schnee';
		17:	str := 'Hagel';
		18:	str := 'Schneeregen';
		19:	str := 'Staub';
		20:	str := 'nebelig';
		21:	str := 'Dunst';
		22:	str := 'rauchig';
		23:	str := 'stürmisch';
		24:	str := 'windig';
		25:	str := 'kalt';
		26:	str := 'bewölkt';
		27:	str := 'meist bewölkt';
		28:	str := 'meist bewölkt';
		29:	str := 'teilweise bewölkt';
		30:	str := 'teilweise bewölkt';
		31:	str := 'klar';
		32:	str := 'sonnig';
		33:	str := 'heiter';
		34:	str := 'heiter';
		35:	str := 'Regen und Hagel';
		36:	str := 'heiß';
		37:	str := 'örtliche Gewitter';
		38:	str := 'vereinzelte Gewitter';
		39:	str := 'vereinzelte Gewitter';
		40:	str := 'vereinzelte Regenfälle';
		41:	str := 'schwere Schneefälle';
		42:	str := 'vereinzelte Schneefälle';
		43:	str := 'schwere Schneefälle';
		44:	str := 'teilweise bewölkt';
		45:	str := 'gewittrige Regenfälle';
		46:	str := 'Schneefälle';
		47:	str := 'örtliche gewittrige Regenfälle';
		ELSE
			str := 'nicht verfügbar';
		END_CASE;
	END_FOR;
END_IF;
act_last := ACTIVATE;

(* revision history
ks	04. may. 2011	rev 1.0
	original version
*)
END_FUNCTION_BLOCK

(* POU YAHOO_WEATHER_ICON_OSCAT, ST *)
FUNCTION_BLOCK YAHOO_WEATHER_ICON_OSCAT
VAR_IN_OUT
	YW : YAHOO_WEATHER_DATA;
END_VAR
VAR_INPUT
	ACTIVATE : BOOL;
END_VAR
VAR
	dat : ARRAY[0..48] OF INT := 4,2,2,4,17,1,3,1,2,2,2,2,2,3,3,3,3,5,3,6,7,14,8,9,9,10,9,11,12,11,12,13,14,15,16,4,14,4,17,2,2,3,3,3,12,2,3,4,0;
	act_last : BOOL;
	x : INT;
END_VAR

(*

version 1.0		04. may. 2011
programmer 		ks
tested by			ks

YAHOO_WEATHER_ICON_OSCAT ändert die ICON Nummer auf den OSCAT-Standard um
*)
IF ACTIVATE AND act_last = FALSE THEN
	x := MIN(YW.CUR_CONDITIONS_CODE,48);
	YW.CUR_CONDITIONS_ICON := dat[x];
	x := MIN(YW.FORCAST_TODAY_CODE,48);
	YW.FORCAST_TODAY_ICON := dat[x];
	x := MIN(YW.FORCAST_TOMORROW_CODE,48);
	YW.FORCAST_TOMORROW_ICON := dat[x];
END_IF;
act_last := ACTIVATE;

(* revision history
ks	04. may. 2011	rev 1.0
	original version
*)
END_FUNCTION_BLOCK

(* POU DLOG_CRON_TAB, ST *)
FUNCTION_BLOCK DLOG_CRON_TAB
VAR_INPUT
	ACTIVATE : BOOL;
	DTI : DT;
	SECOND : STRING(20);
	MINUTE : STRING(20);
	HOUR : STRING(20);
	DAY_OF_MONTH : STRING(20);
	DAY_OF_WEEK : STRING(20);
	MONTH : STRING(20);
END_VAR
VAR_OUTPUT
	Q : BOOL;
END_VAR
VAR
	CD :  DLOG_CRON_DATA;
	activate_old : BOOL;
	datei : DATE;
	dti_last : DT;
	cnt1 : INT;
	cnt2 : INT;
	idx1 : INT;
	idx2 : INT;
	idx3 : INT;
	idx4 : INT;
	pos1 : INT;
	pos2 : INT;
	char_cnt : INT;
	trig_day : BOOL;
	trig_weekday : BOOL;
	str1 : STRING(STRING_LENGTH);
	str2 : STRING(STRING_LENGTH);
	str3 : STRING(STRING_LENGTH);
	num_str1 : STRING(10);
END_VAR

(*
version 1.0		27. oct. 2012
programmer		ks
tested by			ks

DLOG_CRON_TAB erzeugt eine Zeit/Datum Tabelle um damit Ein/Ausschaltvorgänge vorzunehmen
*)
IF ACTIVATE THEN
	IF NOT activate_old THEN
		CD.CE[0].VALUE_MIN := 0;	(* Sekunden *)
		CD.CE[0].VALUE_MAX := 59;
		CD.CE[1].VALUE_MIN := 0;	(* Minuten *)
		CD.CE[1].VALUE_MAX := 59;
		CD.CE[2].VALUE_MIN := 0;	(* Stunden *)
		CD.CE[2].VALUE_MAX := 59;
		CD.CE[3].VALUE_MIN := 1;	(* Tage *)
		CD.CE[3].VALUE_MAX := 31;
		CD.CE[4].VALUE_MIN := 1;	(* Wochentag *)
		CD.CE[4].VALUE_MAX := 7;
		CD.CE[5].VALUE_MIN := 1;	(* Monat *)
		CD.CE[5].VALUE_MAX := 12;

		FOR idx1 := 0 TO 5 DO
			idx3 := CD.CE[idx1].VALUE_MIN;
			idx4 := CD.CE[idx1].VALUE_MAx;
			FOR idx2 := idx3 TO idx4 DO
				CD.CE[idx1].ELEMENTS[idx2] := FALSE;
			END_FOR;
			CD.CE[idx1].ALL_SELECTED := FALSE;
		END_FOR;

		str1 := CONCAT(SECOND,'#');
		str1 := CONCAT(str1,MINUTE);
		str1 := CONCAT(str1,'#');
		str1 := CONCAT(str1,HOUR);
		str1 := CONCAT(str1,'#');
		str1 := CONCAT(str1,DAY_OF_MONTH);
		str1 := CONCAT(str1,'#');
		str1 := CONCAT(str1,DAY_OF_WEEK);
		str1 := CONCAT(str1,'#');
		str1 := CONCAT(str1,MONTH);

		FOR idx1 := 0 TO 5 DO
			str2 := ELEMENT_GET(BYTE#35, idx1, str1);
			IF LEN(str2) > 0 THEN
				cnt1 := ELEMENT_COUNT(BYTE#44, str2);	(* Trenzeichen ',' *)
			ELSE
				cnt1 := 1;
			END_IF;

			FOR idx2 := 0 TO cnt1 -1 DO
				str3 := ELEMENT_GET(BYTE#44, idx2, str2);
				IF FIND(str3, '*/') > 0 AND LEN(str3) <= 10 THEN
					pos1 := DEC_TO_INT(str3);
					IF pos1 > 0 THEN
						idx3 := CD.CE[idx1].VALUE_MIN;
						idx4 := CD.CE[idx1].VALUE_MAX;
						WHILE idx3 <= idx4 DO
							CD.CE[idx1].ELEMENTS[idx3] := TRUE;
							idx3 := idx3 + pos1;
						END_WHILE;
					END_IF;

				ELSE
					IF FIND(str3, '*') > 0 OR LEN(str3) = 0 THEN
						pos1 := CD.CE[idx1].VALUE_MIN;
						pos2 := CD.CE[idx1].VALUE_MAX;
						CD.CE[idx1].ALL_SELECTED := TRUE;
					ELSE
						cnt2 := ELEMENT_COUNT(BYTE#45, str3);	(* Trenzeichen '-' *)
						char_cnt := LEN(str3);
						IF char_cnt >= 1 AND char_cnt <= 10 THEN
							num_str1 := ELEMENT_GET(BYTE#45, 0, str3);
							pos1 := DEC_TO_INT(num_str1);
							pos2 := pos1;
							IF cnt2 = 2 THEN
								num_str1 := ELEMENT_GET(BYTE#45, 1, str3);
								pos2 := DEC_TO_INT(num_str1);
							END_IF;
						END_IF;
					END_IF;

					IF pos1 >= CD.CE[idx1].VALUE_MIN AND pos2 <= CD.CE[idx1].VALUE_MAX THEN
						FOR idx3 := pos1 TO pos2 DO
							CD.CE[idx1].ELEMENTS[idx3] := TRUE;
						END_FOR;
					END_IF;
				END_IF;
			END_FOR;
		END_FOR;
	ELSIF DTI <> dti_last THEN
		CD.CE[0].VALUE := SECOND_OF_DT(DTI); (* Sekunden *)
		CD.CE[1].VALUE := MINUTE_OF_DT(DTI); (* Minuten *)
		CD.CE[2].VALUE := HOUR_OF_DT(DTI); (* Stunden *)
		datei := DT_TO_DATE(DTI);
		CD.CE[3].VALUE := DAY_OF_MONTH(datei); (* Tag *)
		CD.CE[4].VALUE := DAY_OF_WEEK(datei); (* Wochentag *)
		CD.CE[5].VALUE := MONTH_OF_DATE(datei); (*  Monat *)
		dti_last := DTI;

		idx2 := CD.CE[0].VALUE;	(* sekunden *)
		Q := CD.CE[0].ELEMENTS[idx2] = TRUE;
		idx2 := CD.CE[1].VALUE;	(* minuten *)
		Q := Q AND CD.CE[1].ELEMENTS[idx2] = TRUE;
		idx2 := CD.CE[2].VALUE;	(* stunden *)
		Q := Q AND CD.CE[2].ELEMENTS[idx2] = TRUE;
		idx2 := CD.CE[5].VALUE;	(* monat *)
		Q := Q AND CD.CE[5].ELEMENTS[idx2] = TRUE;

		(* auswertung Tag und Wochentag *)
		idx2 := CD.CE[3].VALUE;	(* Tag *)
		trig_day:= CD.CE[3].ELEMENTS[idx2] = TRUE;
		idx2 := CD.CE[4].VALUE;	(* Wochentag *)
		trig_weekday := CD.CE[4].ELEMENTS[idx2] = TRUE;

		IF CD.CE[3].ALL_SELECTED = FALSE AND CD.CE[4].ALL_SELECTED = TRUE THEN
			Q := Q AND trig_day; (* nur Tag auswerten *)
		ELSIF CD.CE[3].ALL_SELECTED = TRUE AND CD.CE[4].ALL_SELECTED = FALSE THEN
			Q := Q AND trig_weekday; (* nur Wochentag auswerten *)
		ELSIF CD.CE[3].ALL_SELECTED = FALSE AND CD.CE[4].ALL_SELECTED = FALSE THEN
			Q := Q AND (trig_weekday OR trig_day); (* Tag und Wochentag auswerten *)
		END_IF;
	END_IF;

END_IF;
activate_old := ACTIVATE;

(* revision history
ks	27. oct. 2011	rev 1.0
	original version
*)
END_FUNCTION_BLOCK

(* POU HTML_DECODE, ST *)
FUNCTION HTML_DECODE : STRING(STRING_LENGTH)
VAR_INPUT
	IN : STRING(STRING_LENGTH);
END_VAR
VAR
	pos : INT;
	end : INT;
	tmp : STRING(10);
	code : STRING(1);
END_VAR

(*
version 1.3		10. may 2010
programmer 	hugo
tested by		oscat

HTML_DECODE converts HTML coded characters to text. 
&amp; is replaced by & ("Ampersand")
&lt; is replaced by < ("lower than")
&gt; is replaced by > ("greater than")
&quot; is replaced by " ("Quote")
all other &names characters are replaced by their respective character codes.

*)
HTML_DECODE := IN;

